FUNCTION "ST10_Flow26_JMagnetLoad&Unload" : Void
VERSION : 1.0
VAR_INPUT
  Enable : BOOL;
END_VAR
VAR_TEMP
  idx : INT;
  tr_cond : ARRAY[1..607] OF BOOL;
  next_active : ARRAY[1..247] OF BOOL;
END_VAR
BEGIN
  IF NOT Enable THEN
    "DB_ST10_Flow26_JMagnetLoad_Unload_State".Flow.Initialized := FALSE;
    FOR idx := 1 TO 247 DO
      "DB_ST10_Flow26_JMagnetLoad_Unload_State".Flow.StepActive[idx] := FALSE;
      "DB_ST10_Flow26_JMagnetLoad_Unload_State".Flow.StepPrev[idx] := FALSE;
    END_FOR;
    "DB_ST10_Flow26_JMagnetLoad_Unload_State".Flow.PalltReleaseRuning := FALSE;
    RETURN;
  END_IF;

  IF NOT "DB_ST10_Flow26_JMagnetLoad_Unload_State".Flow.Initialized THEN
    FOR idx := 1 TO 247 DO
      "DB_ST10_Flow26_JMagnetLoad_Unload_State".Flow.StepActive[idx] := FALSE;
      "DB_ST10_Flow26_JMagnetLoad_Unload_State".Flow.StepPrev[idx] := FALSE;
    END_FOR;
    "DB_ST10_Flow26_JMagnetLoad_Unload_State".Flow.StepActive[1] := TRUE;
    "DB_ST10_Flow26_JMagnetLoad_Unload_State".Flow.StepActive[200] := TRUE;
    "DB_ST10_Flow26_JMagnetLoad_Unload_State".Flow.Initialized := TRUE;
  END_IF;


  IF "DB_ST10_Flow26_JMagnetLoad_Unload_State".Flow.StepActive[119] THEN
    "DB_ST10_Flow26_JMagnetLoad_Unload_State".Flow.StepTime.AriveTimeDelay_1 := "DB_ST10_Flow26_JMagnetLoad_Unload_State".Flow.StepTime.AriveTimeDelay_1 + OB1_PREV_CYCLE;
  ELSE
    "DB_ST10_Flow26_JMagnetLoad_Unload_State".Flow.StepTime.AriveTimeDelay_1 := T#0S;
  END_IF;
  IF "DB_ST10_Flow26_JMagnetLoad_Unload_State".Flow.StepActive[168] THEN
    "DB_ST10_Flow26_JMagnetLoad_Unload_State".Flow.StepTime.AriveTimeDelay_10 := "DB_ST10_Flow26_JMagnetLoad_Unload_State".Flow.StepTime.AriveTimeDelay_10 + OB1_PREV_CYCLE;
  ELSE
    "DB_ST10_Flow26_JMagnetLoad_Unload_State".Flow.StepTime.AriveTimeDelay_10 := T#0S;
  END_IF;
  IF "DB_ST10_Flow26_JMagnetLoad_Unload_State".Flow.StepActive[173] THEN
    "DB_ST10_Flow26_JMagnetLoad_Unload_State".Flow.StepTime.AriveTimeDelay_11 := "DB_ST10_Flow26_JMagnetLoad_Unload_State".Flow.StepTime.AriveTimeDelay_11 + OB1_PREV_CYCLE;
  ELSE
    "DB_ST10_Flow26_JMagnetLoad_Unload_State".Flow.StepTime.AriveTimeDelay_11 := T#0S;
  END_IF;
  IF "DB_ST10_Flow26_JMagnetLoad_Unload_State".Flow.StepActive[120] THEN
    "DB_ST10_Flow26_JMagnetLoad_Unload_State".Flow.StepTime.AriveTimeDelay_2 := "DB_ST10_Flow26_JMagnetLoad_Unload_State".Flow.StepTime.AriveTimeDelay_2 + OB1_PREV_CYCLE;
  ELSE
    "DB_ST10_Flow26_JMagnetLoad_Unload_State".Flow.StepTime.AriveTimeDelay_2 := T#0S;
  END_IF;
  IF "DB_ST10_Flow26_JMagnetLoad_Unload_State".Flow.StepActive[125] THEN
    "DB_ST10_Flow26_JMagnetLoad_Unload_State".Flow.StepTime.AriveTimeDelay_3 := "DB_ST10_Flow26_JMagnetLoad_Unload_State".Flow.StepTime.AriveTimeDelay_3 + OB1_PREV_CYCLE;
  ELSE
    "DB_ST10_Flow26_JMagnetLoad_Unload_State".Flow.StepTime.AriveTimeDelay_3 := T#0S;
  END_IF;
  IF "DB_ST10_Flow26_JMagnetLoad_Unload_State".Flow.StepActive[130] THEN
    "DB_ST10_Flow26_JMagnetLoad_Unload_State".Flow.StepTime.AriveTimeDelay_4 := "DB_ST10_Flow26_JMagnetLoad_Unload_State".Flow.StepTime.AriveTimeDelay_4 + OB1_PREV_CYCLE;
  ELSE
    "DB_ST10_Flow26_JMagnetLoad_Unload_State".Flow.StepTime.AriveTimeDelay_4 := T#0S;
  END_IF;
  IF "DB_ST10_Flow26_JMagnetLoad_Unload_State".Flow.StepActive[136] THEN
    "DB_ST10_Flow26_JMagnetLoad_Unload_State".Flow.StepTime.AriveTimeDelay_5 := "DB_ST10_Flow26_JMagnetLoad_Unload_State".Flow.StepTime.AriveTimeDelay_5 + OB1_PREV_CYCLE;
  ELSE
    "DB_ST10_Flow26_JMagnetLoad_Unload_State".Flow.StepTime.AriveTimeDelay_5 := T#0S;
  END_IF;
  IF "DB_ST10_Flow26_JMagnetLoad_Unload_State".Flow.StepActive[141] THEN
    "DB_ST10_Flow26_JMagnetLoad_Unload_State".Flow.StepTime.AriveTimeDelay_6 := "DB_ST10_Flow26_JMagnetLoad_Unload_State".Flow.StepTime.AriveTimeDelay_6 + OB1_PREV_CYCLE;
  ELSE
    "DB_ST10_Flow26_JMagnetLoad_Unload_State".Flow.StepTime.AriveTimeDelay_6 := T#0S;
  END_IF;
  IF "DB_ST10_Flow26_JMagnetLoad_Unload_State".Flow.StepActive[148] THEN
    "DB_ST10_Flow26_JMagnetLoad_Unload_State".Flow.StepTime.AriveTimeDelay_7 := "DB_ST10_Flow26_JMagnetLoad_Unload_State".Flow.StepTime.AriveTimeDelay_7 + OB1_PREV_CYCLE;
  ELSE
    "DB_ST10_Flow26_JMagnetLoad_Unload_State".Flow.StepTime.AriveTimeDelay_7 := T#0S;
  END_IF;
  IF "DB_ST10_Flow26_JMagnetLoad_Unload_State".Flow.StepActive[159] THEN
    "DB_ST10_Flow26_JMagnetLoad_Unload_State".Flow.StepTime.AriveTimeDelay_8 := "DB_ST10_Flow26_JMagnetLoad_Unload_State".Flow.StepTime.AriveTimeDelay_8 + OB1_PREV_CYCLE;
  ELSE
    "DB_ST10_Flow26_JMagnetLoad_Unload_State".Flow.StepTime.AriveTimeDelay_8 := T#0S;
  END_IF;
  IF "DB_ST10_Flow26_JMagnetLoad_Unload_State".Flow.StepActive[163] THEN
    "DB_ST10_Flow26_JMagnetLoad_Unload_State".Flow.StepTime.AriveTimeDelay_9 := "DB_ST10_Flow26_JMagnetLoad_Unload_State".Flow.StepTime.AriveTimeDelay_9 + OB1_PREV_CYCLE;
  ELSE
    "DB_ST10_Flow26_JMagnetLoad_Unload_State".Flow.StepTime.AriveTimeDelay_9 := T#0S;
  END_IF;
  IF "DB_ST10_Flow26_JMagnetLoad_Unload_State".Flow.StepActive[31] THEN
    "DB_ST10_Flow26_JMagnetLoad_Unload_State".Flow.StepTime.CheckPalletExist := "DB_ST10_Flow26_JMagnetLoad_Unload_State".Flow.StepTime.CheckPalletExist + OB1_PREV_CYCLE;
  ELSE
    "DB_ST10_Flow26_JMagnetLoad_Unload_State".Flow.StepTime.CheckPalletExist := T#0S;
  END_IF;
  IF "DB_ST10_Flow26_JMagnetLoad_Unload_State".Flow.StepActive[32] THEN
    "DB_ST10_Flow26_JMagnetLoad_Unload_State".Flow.StepTime.CheckPalletExist_1 := "DB_ST10_Flow26_JMagnetLoad_Unload_State".Flow.StepTime.CheckPalletExist_1 + OB1_PREV_CYCLE;
  ELSE
    "DB_ST10_Flow26_JMagnetLoad_Unload_State".Flow.StepTime.CheckPalletExist_1 := T#0S;
  END_IF;
  IF "DB_ST10_Flow26_JMagnetLoad_Unload_State".Flow.StepActive[76] THEN
    "DB_ST10_Flow26_JMagnetLoad_Unload_State".Flow.StepTime.CheckPalletExist_10 := "DB_ST10_Flow26_JMagnetLoad_Unload_State".Flow.StepTime.CheckPalletExist_10 + OB1_PREV_CYCLE;
  ELSE
    "DB_ST10_Flow26_JMagnetLoad_Unload_State".Flow.StepTime.CheckPalletExist_10 := T#0S;
  END_IF;
  IF "DB_ST10_Flow26_JMagnetLoad_Unload_State".Flow.StepActive[41] THEN
    "DB_ST10_Flow26_JMagnetLoad_Unload_State".Flow.StepTime.CheckPalletExist_2 := "DB_ST10_Flow26_JMagnetLoad_Unload_State".Flow.StepTime.CheckPalletExist_2 + OB1_PREV_CYCLE;
  ELSE
    "DB_ST10_Flow26_JMagnetLoad_Unload_State".Flow.StepTime.CheckPalletExist_2 := T#0S;
  END_IF;
  IF "DB_ST10_Flow26_JMagnetLoad_Unload_State".Flow.StepActive[45] THEN
    "DB_ST10_Flow26_JMagnetLoad_Unload_State".Flow.StepTime.CheckPalletExist_3 := "DB_ST10_Flow26_JMagnetLoad_Unload_State".Flow.StepTime.CheckPalletExist_3 + OB1_PREV_CYCLE;
  ELSE
    "DB_ST10_Flow26_JMagnetLoad_Unload_State".Flow.StepTime.CheckPalletExist_3 := T#0S;
  END_IF;
  IF "DB_ST10_Flow26_JMagnetLoad_Unload_State".Flow.StepActive[49] THEN
    "DB_ST10_Flow26_JMagnetLoad_Unload_State".Flow.StepTime.CheckPalletExist_4 := "DB_ST10_Flow26_JMagnetLoad_Unload_State".Flow.StepTime.CheckPalletExist_4 + OB1_PREV_CYCLE;
  ELSE
    "DB_ST10_Flow26_JMagnetLoad_Unload_State".Flow.StepTime.CheckPalletExist_4 := T#0S;
  END_IF;
  IF "DB_ST10_Flow26_JMagnetLoad_Unload_State".Flow.StepActive[53] THEN
    "DB_ST10_Flow26_JMagnetLoad_Unload_State".Flow.StepTime.CheckPalletExist_5 := "DB_ST10_Flow26_JMagnetLoad_Unload_State".Flow.StepTime.CheckPalletExist_5 + OB1_PREV_CYCLE;
  ELSE
    "DB_ST10_Flow26_JMagnetLoad_Unload_State".Flow.StepTime.CheckPalletExist_5 := T#0S;
  END_IF;
  IF "DB_ST10_Flow26_JMagnetLoad_Unload_State".Flow.StepActive[57] THEN
    "DB_ST10_Flow26_JMagnetLoad_Unload_State".Flow.StepTime.CheckPalletExist_6 := "DB_ST10_Flow26_JMagnetLoad_Unload_State".Flow.StepTime.CheckPalletExist_6 + OB1_PREV_CYCLE;
  ELSE
    "DB_ST10_Flow26_JMagnetLoad_Unload_State".Flow.StepTime.CheckPalletExist_6 := T#0S;
  END_IF;
  IF "DB_ST10_Flow26_JMagnetLoad_Unload_State".Flow.StepActive[64] THEN
    "DB_ST10_Flow26_JMagnetLoad_Unload_State".Flow.StepTime.CheckPalletExist_7 := "DB_ST10_Flow26_JMagnetLoad_Unload_State".Flow.StepTime.CheckPalletExist_7 + OB1_PREV_CYCLE;
  ELSE
    "DB_ST10_Flow26_JMagnetLoad_Unload_State".Flow.StepTime.CheckPalletExist_7 := T#0S;
  END_IF;
  IF "DB_ST10_Flow26_JMagnetLoad_Unload_State".Flow.StepActive[68] THEN
    "DB_ST10_Flow26_JMagnetLoad_Unload_State".Flow.StepTime.CheckPalletExist_8 := "DB_ST10_Flow26_JMagnetLoad_Unload_State".Flow.StepTime.CheckPalletExist_8 + OB1_PREV_CYCLE;
  ELSE
    "DB_ST10_Flow26_JMagnetLoad_Unload_State".Flow.StepTime.CheckPalletExist_8 := T#0S;
  END_IF;
  IF "DB_ST10_Flow26_JMagnetLoad_Unload_State".Flow.StepActive[72] THEN
    "DB_ST10_Flow26_JMagnetLoad_Unload_State".Flow.StepTime.CheckPalletExist_9 := "DB_ST10_Flow26_JMagnetLoad_Unload_State".Flow.StepTime.CheckPalletExist_9 + OB1_PREV_CYCLE;
  ELSE
    "DB_ST10_Flow26_JMagnetLoad_Unload_State".Flow.StepTime.CheckPalletExist_9 := T#0S;
  END_IF;
  IF "DB_ST10_Flow26_JMagnetLoad_Unload_State".Flow.StepActive[160] THEN
    "DB_ST10_Flow26_JMagnetLoad_Unload_State".Flow.StepTime.LoadStop_11 := "DB_ST10_Flow26_JMagnetLoad_Unload_State".Flow.StepTime.LoadStop_11 + OB1_PREV_CYCLE;
  ELSE
    "DB_ST10_Flow26_JMagnetLoad_Unload_State".Flow.StepTime.LoadStop_11 := T#0S;
  END_IF;
  IF "DB_ST10_Flow26_JMagnetLoad_Unload_State".Flow.StepActive[62] THEN
    "DB_ST10_Flow26_JMagnetLoad_Unload_State".Flow.StepTime.LoadStop_12 := "DB_ST10_Flow26_JMagnetLoad_Unload_State".Flow.StepTime.LoadStop_12 + OB1_PREV_CYCLE;
  ELSE
    "DB_ST10_Flow26_JMagnetLoad_Unload_State".Flow.StepTime.LoadStop_12 := T#0S;
  END_IF;
  IF "DB_ST10_Flow26_JMagnetLoad_Unload_State".Flow.StepActive[63] THEN
    "DB_ST10_Flow26_JMagnetLoad_Unload_State".Flow.StepTime.LoadStop_13 := "DB_ST10_Flow26_JMagnetLoad_Unload_State".Flow.StepTime.LoadStop_13 + OB1_PREV_CYCLE;
  ELSE
    "DB_ST10_Flow26_JMagnetLoad_Unload_State".Flow.StepTime.LoadStop_13 := T#0S;
  END_IF;
  IF "DB_ST10_Flow26_JMagnetLoad_Unload_State".Flow.StepActive[61] THEN
    "DB_ST10_Flow26_JMagnetLoad_Unload_State".Flow.StepTime.LoadStop_14 := "DB_ST10_Flow26_JMagnetLoad_Unload_State".Flow.StepTime.LoadStop_14 + OB1_PREV_CYCLE;
  ELSE
    "DB_ST10_Flow26_JMagnetLoad_Unload_State".Flow.StepTime.LoadStop_14 := T#0S;
  END_IF;
  IF "DB_ST10_Flow26_JMagnetLoad_Unload_State".Flow.StepActive[25] THEN
    "DB_ST10_Flow26_JMagnetLoad_Unload_State".Flow.StepTime.MotorRunDelay := "DB_ST10_Flow26_JMagnetLoad_Unload_State".Flow.StepTime.MotorRunDelay + OB1_PREV_CYCLE;
  ELSE
    "DB_ST10_Flow26_JMagnetLoad_Unload_State".Flow.StepTime.MotorRunDelay := T#0S;
  END_IF;
  IF "DB_ST10_Flow26_JMagnetLoad_Unload_State".Flow.StepActive[26] THEN
    "DB_ST10_Flow26_JMagnetLoad_Unload_State".Flow.StepTime.MotorRunDelay_1 := "DB_ST10_Flow26_JMagnetLoad_Unload_State".Flow.StepTime.MotorRunDelay_1 + OB1_PREV_CYCLE;
  ELSE
    "DB_ST10_Flow26_JMagnetLoad_Unload_State".Flow.StepTime.MotorRunDelay_1 := T#0S;
  END_IF;
  IF "DB_ST10_Flow26_JMagnetLoad_Unload_State".Flow.StepActive[118] THEN
    "DB_ST10_Flow26_JMagnetLoad_Unload_State".Flow.StepTime.StoperRelease_1 := "DB_ST10_Flow26_JMagnetLoad_Unload_State".Flow.StepTime.StoperRelease_1 + OB1_PREV_CYCLE;
  ELSE
    "DB_ST10_Flow26_JMagnetLoad_Unload_State".Flow.StepTime.StoperRelease_1 := T#0S;
  END_IF;
  IF "DB_ST10_Flow26_JMagnetLoad_Unload_State".Flow.StepActive[170] THEN
    "DB_ST10_Flow26_JMagnetLoad_Unload_State".Flow.StepTime.StoperRelease_10 := "DB_ST10_Flow26_JMagnetLoad_Unload_State".Flow.StepTime.StoperRelease_10 + OB1_PREV_CYCLE;
  ELSE
    "DB_ST10_Flow26_JMagnetLoad_Unload_State".Flow.StepTime.StoperRelease_10 := T#0S;
  END_IF;
  IF "DB_ST10_Flow26_JMagnetLoad_Unload_State".Flow.StepActive[175] THEN
    "DB_ST10_Flow26_JMagnetLoad_Unload_State".Flow.StepTime.StoperRelease_11 := "DB_ST10_Flow26_JMagnetLoad_Unload_State".Flow.StepTime.StoperRelease_11 + OB1_PREV_CYCLE;
  ELSE
    "DB_ST10_Flow26_JMagnetLoad_Unload_State".Flow.StepTime.StoperRelease_11 := T#0S;
  END_IF;
  IF "DB_ST10_Flow26_JMagnetLoad_Unload_State".Flow.StepActive[122] THEN
    "DB_ST10_Flow26_JMagnetLoad_Unload_State".Flow.StepTime.StoperRelease_2 := "DB_ST10_Flow26_JMagnetLoad_Unload_State".Flow.StepTime.StoperRelease_2 + OB1_PREV_CYCLE;
  ELSE
    "DB_ST10_Flow26_JMagnetLoad_Unload_State".Flow.StepTime.StoperRelease_2 := T#0S;
  END_IF;
  IF "DB_ST10_Flow26_JMagnetLoad_Unload_State".Flow.StepActive[127] THEN
    "DB_ST10_Flow26_JMagnetLoad_Unload_State".Flow.StepTime.StoperRelease_3 := "DB_ST10_Flow26_JMagnetLoad_Unload_State".Flow.StepTime.StoperRelease_3 + OB1_PREV_CYCLE;
  ELSE
    "DB_ST10_Flow26_JMagnetLoad_Unload_State".Flow.StepTime.StoperRelease_3 := T#0S;
  END_IF;
  IF "DB_ST10_Flow26_JMagnetLoad_Unload_State".Flow.StepActive[133] THEN
    "DB_ST10_Flow26_JMagnetLoad_Unload_State".Flow.StepTime.StoperRelease_4 := "DB_ST10_Flow26_JMagnetLoad_Unload_State".Flow.StepTime.StoperRelease_4 + OB1_PREV_CYCLE;
  ELSE
    "DB_ST10_Flow26_JMagnetLoad_Unload_State".Flow.StepTime.StoperRelease_4 := T#0S;
  END_IF;
  IF "DB_ST10_Flow26_JMagnetLoad_Unload_State".Flow.StepActive[138] THEN
    "DB_ST10_Flow26_JMagnetLoad_Unload_State".Flow.StepTime.StoperRelease_5 := "DB_ST10_Flow26_JMagnetLoad_Unload_State".Flow.StepTime.StoperRelease_5 + OB1_PREV_CYCLE;
  ELSE
    "DB_ST10_Flow26_JMagnetLoad_Unload_State".Flow.StepTime.StoperRelease_5 := T#0S;
  END_IF;
  IF "DB_ST10_Flow26_JMagnetLoad_Unload_State".Flow.StepActive[145] THEN
    "DB_ST10_Flow26_JMagnetLoad_Unload_State".Flow.StepTime.StoperRelease_6 := "DB_ST10_Flow26_JMagnetLoad_Unload_State".Flow.StepTime.StoperRelease_6 + OB1_PREV_CYCLE;
  ELSE
    "DB_ST10_Flow26_JMagnetLoad_Unload_State".Flow.StepTime.StoperRelease_6 := T#0S;
  END_IF;
  IF "DB_ST10_Flow26_JMagnetLoad_Unload_State".Flow.StepActive[150] THEN
    "DB_ST10_Flow26_JMagnetLoad_Unload_State".Flow.StepTime.StoperRelease_7 := "DB_ST10_Flow26_JMagnetLoad_Unload_State".Flow.StepTime.StoperRelease_7 + OB1_PREV_CYCLE;
  ELSE
    "DB_ST10_Flow26_JMagnetLoad_Unload_State".Flow.StepTime.StoperRelease_7 := T#0S;
  END_IF;
  IF "DB_ST10_Flow26_JMagnetLoad_Unload_State".Flow.StepActive[162] THEN
    "DB_ST10_Flow26_JMagnetLoad_Unload_State".Flow.StepTime.StoperRelease_8 := "DB_ST10_Flow26_JMagnetLoad_Unload_State".Flow.StepTime.StoperRelease_8 + OB1_PREV_CYCLE;
  ELSE
    "DB_ST10_Flow26_JMagnetLoad_Unload_State".Flow.StepTime.StoperRelease_8 := T#0S;
  END_IF;
  IF "DB_ST10_Flow26_JMagnetLoad_Unload_State".Flow.StepActive[165] THEN
    "DB_ST10_Flow26_JMagnetLoad_Unload_State".Flow.StepTime.StoperRelease_9 := "DB_ST10_Flow26_JMagnetLoad_Unload_State".Flow.StepTime.StoperRelease_9 + OB1_PREV_CYCLE;
  ELSE
    "DB_ST10_Flow26_JMagnetLoad_Unload_State".Flow.StepTime.StoperRelease_9 := T#0S;
  END_IF;
  IF "DB_ST10_Flow26_JMagnetLoad_Unload_State".Flow.StepActive[116] THEN
    "DB_ST10_Flow26_JMagnetLoad_Unload_State".Flow.StepTime.StoperReset := "DB_ST10_Flow26_JMagnetLoad_Unload_State".Flow.StepTime.StoperReset + OB1_PREV_CYCLE;
  ELSE
    "DB_ST10_Flow26_JMagnetLoad_Unload_State".Flow.StepTime.StoperReset := T#0S;
  END_IF;
  IF "DB_ST10_Flow26_JMagnetLoad_Unload_State".Flow.StepActive[124] THEN
    "DB_ST10_Flow26_JMagnetLoad_Unload_State".Flow.StepTime.TimeDelay := "DB_ST10_Flow26_JMagnetLoad_Unload_State".Flow.StepTime.TimeDelay + OB1_PREV_CYCLE;
  ELSE
    "DB_ST10_Flow26_JMagnetLoad_Unload_State".Flow.StepTime.TimeDelay := T#0S;
  END_IF;
  IF "DB_ST10_Flow26_JMagnetLoad_Unload_State".Flow.StepActive[129] THEN
    "DB_ST10_Flow26_JMagnetLoad_Unload_State".Flow.StepTime.TimeDelay_1 := "DB_ST10_Flow26_JMagnetLoad_Unload_State".Flow.StepTime.TimeDelay_1 + OB1_PREV_CYCLE;
  ELSE
    "DB_ST10_Flow26_JMagnetLoad_Unload_State".Flow.StepTime.TimeDelay_1 := T#0S;
  END_IF;
  IF "DB_ST10_Flow26_JMagnetLoad_Unload_State".Flow.StepActive[135] THEN
    "DB_ST10_Flow26_JMagnetLoad_Unload_State".Flow.StepTime.TimeDelay_2 := "DB_ST10_Flow26_JMagnetLoad_Unload_State".Flow.StepTime.TimeDelay_2 + OB1_PREV_CYCLE;
  ELSE
    "DB_ST10_Flow26_JMagnetLoad_Unload_State".Flow.StepTime.TimeDelay_2 := T#0S;
  END_IF;
  IF "DB_ST10_Flow26_JMagnetLoad_Unload_State".Flow.StepActive[140] THEN
    "DB_ST10_Flow26_JMagnetLoad_Unload_State".Flow.StepTime.TimeDelay_3 := "DB_ST10_Flow26_JMagnetLoad_Unload_State".Flow.StepTime.TimeDelay_3 + OB1_PREV_CYCLE;
  ELSE
    "DB_ST10_Flow26_JMagnetLoad_Unload_State".Flow.StepTime.TimeDelay_3 := T#0S;
  END_IF;
  IF "DB_ST10_Flow26_JMagnetLoad_Unload_State".Flow.StepActive[147] THEN
    "DB_ST10_Flow26_JMagnetLoad_Unload_State".Flow.StepTime.TimeDelay_4 := "DB_ST10_Flow26_JMagnetLoad_Unload_State".Flow.StepTime.TimeDelay_4 + OB1_PREV_CYCLE;
  ELSE
    "DB_ST10_Flow26_JMagnetLoad_Unload_State".Flow.StepTime.TimeDelay_4 := T#0S;
  END_IF;
  IF "DB_ST10_Flow26_JMagnetLoad_Unload_State".Flow.StepActive[152] THEN
    "DB_ST10_Flow26_JMagnetLoad_Unload_State".Flow.StepTime.TimeDelay_5 := "DB_ST10_Flow26_JMagnetLoad_Unload_State".Flow.StepTime.TimeDelay_5 + OB1_PREV_CYCLE;
  ELSE
    "DB_ST10_Flow26_JMagnetLoad_Unload_State".Flow.StepTime.TimeDelay_5 := T#0S;
  END_IF;
  IF "DB_ST10_Flow26_JMagnetLoad_Unload_State".Flow.StepActive[167] THEN
    "DB_ST10_Flow26_JMagnetLoad_Unload_State".Flow.StepTime.TimeDelay_6 := "DB_ST10_Flow26_JMagnetLoad_Unload_State".Flow.StepTime.TimeDelay_6 + OB1_PREV_CYCLE;
  ELSE
    "DB_ST10_Flow26_JMagnetLoad_Unload_State".Flow.StepTime.TimeDelay_6 := T#0S;
  END_IF;
  IF "DB_ST10_Flow26_JMagnetLoad_Unload_State".Flow.StepActive[172] THEN
    "DB_ST10_Flow26_JMagnetLoad_Unload_State".Flow.StepTime.TimeDelay_7 := "DB_ST10_Flow26_JMagnetLoad_Unload_State".Flow.StepTime.TimeDelay_7 + OB1_PREV_CYCLE;
  ELSE
    "DB_ST10_Flow26_JMagnetLoad_Unload_State".Flow.StepTime.TimeDelay_7 := T#0S;
  END_IF;
  IF "DB_ST10_Flow26_JMagnetLoad_Unload_State".Flow.StepActive[177] THEN
    "DB_ST10_Flow26_JMagnetLoad_Unload_State".Flow.StepTime.TimeDelay_8 := "DB_ST10_Flow26_JMagnetLoad_Unload_State".Flow.StepTime.TimeDelay_8 + OB1_PREV_CYCLE;
  ELSE
    "DB_ST10_Flow26_JMagnetLoad_Unload_State".Flow.StepTime.TimeDelay_8 := T#0S;
  END_IF;
  IF "DB_ST10_Flow26_JMagnetLoad_Unload_State".Flow.StepActive[184] THEN
    "DB_ST10_Flow26_JMagnetLoad_Unload_State".Flow.StepTime.TimeDelay_9 := "DB_ST10_Flow26_JMagnetLoad_Unload_State".Flow.StepTime.TimeDelay_9 + OB1_PREV_CYCLE;
  ELSE
    "DB_ST10_Flow26_JMagnetLoad_Unload_State".Flow.StepTime.TimeDelay_9 := T#0S;
  END_IF;

  tr_cond[1] := (TRUE) AND ("DB_ST10_Flow26_JMagnetLoad_Unload_State".Flow.iSysInface.Ready);
  tr_cond[2] := TRUE;
  tr_cond[3] := TRUE;
  tr_cond[10] := TRUE;
  tr_cond[27] := TRUE;
  tr_cond[28] := TRUE;
  tr_cond[29] := ("DB_ST10_Flow26_JMagnetLoad_Unload_State".Flow.StepTime.MotorRunDelay) > (t#5000MS);
  tr_cond[30] := TRUE;
  tr_cond[31] := ("DB_ST10_Flow26_JMagnetLoad_Unload_State".Flow.StepTime.MotorRunDelay_1) > (t#5000MS);
  tr_cond[32] := ("DB_ST10_Flow26_JMagnetLoad_Unload_State".Flow.StepTime.CheckPalletExist_7) > (t#1000MS);
  tr_cond[33] := TRUE;
  tr_cond[34] := (("DB_ST10_Flow26_JMagnetLoad_Unload_State".Flow.StepTime.CheckPalletExist) > (t#1000MS)) AND (NOT ("DB_ST10_Flow26_JMagnetLoad_Unload_State".AutoProcessControl.Robot_1.ClearPart));
  tr_cond[35] := ("DB_ST10_Flow26_JMagnetLoad_Unload_State".Flow.StepTime.CheckPalletExist_1) > (t#1000MS);
  tr_cond[36] := ("DB_ST10_Flow26_JMagnetLoad_Unload_State".Flow.StepTime.CheckPalletExist_2) > (t#1000MS);
  tr_cond[37] := ((TRUE) AND (MotorControl.Dev[13].OutControl.o_Ready)) AND (MotorControl.Dev[14].OutControl.o_Ready);
  tr_cond[38] := TRUE;
  tr_cond[39] := (TRUE) AND (MotorControl.Dev[13].OutControl.o_Ready);
  tr_cond[40] := (TRUE) AND ("DB_ST10_Flow26_JMagnetLoad_Unload_State".AutoProcessControl.Global.J.LoadStopRequestPallet_1);
  tr_cond[41] := ((TRUE) AND (iJ-magnetLoadingDetection2)) OR ((TRUE) AND ("DB_ST10_Flow26_JMagnetLoad_Unload_State".AutoProcessControl.Global.J.EmptyPallet));
  tr_cond[42] := ((TRUE) AND (iJ-magnetLoadingDetection3)) OR ((TRUE) AND ("DB_ST10_Flow26_JMagnetLoad_Unload_State".AutoProcessControl.Global.J.EmptyPallet));
  tr_cond[43] := (TRUE) AND (MotorControl.Dev[13].OutControl.o_Ready);
  tr_cond[44] := (TRUE) AND ("DB_ST10_Flow26_JMagnetLoad_Unload_State".AutoProcessControl.Global.J.LoadStopRequestPallet_2);
  tr_cond[45] := ((TRUE) AND (iJ-magnetLoadingDetection4)) OR ((TRUE) AND ("DB_ST10_Flow26_JMagnetLoad_Unload_State".AutoProcessControl.Global.J.EmptyPallet));
  tr_cond[46] := (TRUE) AND (MotorControl.Dev[13].OutControl.o_Ready);
  tr_cond[47] := (TRUE) AND ("DB_ST10_Flow26_JMagnetLoad_Unload_State".AutoProcessControl.Global.J.LoadStopRequestPallet_3);
  tr_cond[48] := (((TRUE) AND (iJ-magnetLiftingPalletDischargeDetection)) AND (NOT (iJ-MagnetMiddleDetection))) OR ((TRUE) AND ("DB_ST10_Flow26_JMagnetLoad_Unload_State".AutoProcessControl.Global.J.EmptyPallet));
  tr_cond[49] := ("DB_ST10_Flow26_JMagnetLoad_Unload_State".Flow.StepTime.CheckPalletExist_3) > (t#1000MS);
  tr_cond[50] := (TRUE) AND (MotorControl.Dev[13].OutControl.o_Ready);
  tr_cond[51] := (TRUE) AND ("DB_ST10_Flow26_JMagnetLoad_Unload_State".AutoProcessControl.Global.J.LoadStopRequestPallet_4);
  tr_cond[52] := (TRUE) AND (iJ-magnetTakeDetection2);
  tr_cond[53] := ("DB_ST10_Flow26_JMagnetLoad_Unload_State".Flow.StepTime.CheckPalletExist_4) > (t#1000MS);
  tr_cond[54] := (TRUE) AND (MotorControl.Dev[14].OutControl.o_Ready);
  tr_cond[55] := (TRUE) AND ("DB_ST10_Flow26_JMagnetLoad_Unload_State".AutoProcessControl.Global.J.EmptyStopRequestPallet_2);
  tr_cond[56] := (TRUE) AND (iJ-magnetTakeDetection3);
  tr_cond[57] := ("DB_ST10_Flow26_JMagnetLoad_Unload_State".Flow.StepTime.CheckPalletExist_5) > (t#1000MS);
  tr_cond[58] := (TRUE) AND (MotorControl.Dev[14].OutControl.o_Ready);
  tr_cond[59] := (TRUE) AND ("DB_ST10_Flow26_JMagnetLoad_Unload_State".AutoProcessControl.Global.J.EmptyStopRequestPallet_3);
  tr_cond[60] := (TRUE) AND (iJ-magnetTakeShaftDetection);
  tr_cond[61] := ("DB_ST10_Flow26_JMagnetLoad_Unload_State".Flow.StepTime.CheckPalletExist_6) > (t#1000MS);
  tr_cond[62] := (TRUE) AND (MotorControl.Dev[14].OutControl.o_Ready);
  tr_cond[63] := (TRUE) AND (NOT (iJ-magnetTakeShaftDetection));
  tr_cond[64] := ((TRUE) AND (iJ-magnetTakeGateDetection)) OR ((TRUE) AND (NOT ("DB_ST10_Flow26_JMagnetLoad_Unload_State".AutoProcessControl.Global.J.EmptyPallet)));
  tr_cond[65] := ("DB_ST10_Flow26_JMagnetLoad_Unload_State".Flow.StepTime.CheckPalletExist_7) > (t#1000MS);
  tr_cond[66] := (TRUE) AND (MotorControl.Dev[13].OutControl.o_Ready);
  tr_cond[67] := (TRUE) AND (NOT (iJ-magnetTakeGateDetection));
  tr_cond[68] := (TRUE) AND (J-mganePalletEmptyCheck1);
  tr_cond[69] := ("DB_ST10_Flow26_JMagnetLoad_Unload_State".Flow.StepTime.CheckPalletExist_8) > (t#1000MS);
  tr_cond[70] := (TRUE) AND (MotorControl.Dev[13].OutControl.o_Ready);
  tr_cond[71] := (TRUE) AND ("DB_ST10_Flow26_JMagnetLoad_Unload_State".AutoProcessControl.Global.J.LoadStopRequestPallet_2);
  tr_cond[72] := (TRUE) AND (J-mganePalletEmptyCheck2);
  tr_cond[73] := ("DB_ST10_Flow26_JMagnetLoad_Unload_State".Flow.StepTime.CheckPalletExist_9) > (t#1000MS);
  tr_cond[74] := (TRUE) AND (MotorControl.Dev[13].OutControl.o_Ready);
  tr_cond[75] := (TRUE) AND ("DB_ST10_Flow26_JMagnetLoad_Unload_State".AutoProcessControl.Global.J.LoadStopRequestPallet_3);
  tr_cond[76] := (TRUE) AND (J-mganePalletEmptyCheck3);
  tr_cond[77] := ("DB_ST10_Flow26_JMagnetLoad_Unload_State".Flow.StepTime.CheckPalletExist_10) > (t#1000MS);
  tr_cond[78] := (TRUE) AND (MotorControl.Dev[13].OutControl.o_Ready);
  tr_cond[79] := (TRUE) AND ("DB_ST10_Flow26_JMagnetLoad_Unload_State".AutoProcessControl.Global.J.LoadStopRequestPallet_4);
  tr_cond[80] := TRUE;
  tr_cond[81] := (TRUE) AND (NOT (iJ-MagnetMiddleDetection));
  tr_cond[100] := TRUE;
  tr_cond[116] := ("DB_ST10_Flow26_JMagnetLoad_Unload_State".Flow.StepTime.StoperReset) > (t#1000MS);
  tr_cond[117] := TRUE;
  tr_cond[118] := ("DB_ST10_Flow26_JMagnetLoad_Unload_State".Flow.StepTime.StoperRelease_1) > (t#1000MS);
  tr_cond[119] := ("DB_ST10_Flow26_JMagnetLoad_Unload_State".Flow.StepTime.AriveTimeDelay_1) > (t#500MS);
  tr_cond[120] := TRUE;
  tr_cond[121] := TRUE;
  tr_cond[122] := TRUE;
  tr_cond[123] := ("DB_ST10_Flow26_JMagnetLoad_Unload_State".Flow.StepTime.AriveTimeDelay_2) > (t#500MS);
  tr_cond[124] := TRUE;
  tr_cond[125] := ("DB_ST10_Flow26_JMagnetLoad_Unload_State".Flow.StepTime.StoperRelease_2) > (t#1000MS);
  tr_cond[126] := ("DB_ST10_Flow26_JMagnetLoad_Unload_State".Flow.StepTime.CheckPalletExist_1) > (t#1000MS);
  tr_cond[127] := ((TRUE) AND (iJ-magnetLoadingDetection2)) OR ((TRUE) AND ("DB_ST10_Flow26_JMagnetLoad_Unload_State".AutoProcessControl.Global.J.EmptyPallet));
  tr_cond[128] := ("DB_ST10_Flow26_JMagnetLoad_Unload_State".Flow.StepTime.TimeDelay) > (t#500MS);
  tr_cond[129] := ("DB_ST10_Flow26_JMagnetLoad_Unload_State".Flow.StepTime.AriveTimeDelay_3) > (t#500MS);
  tr_cond[130] := TRUE;
  tr_cond[131] := ("DB_ST10_Flow26_JMagnetLoad_Unload_State".Flow.StepTime.StoperRelease_3) > (t#1000MS);
  tr_cond[132] := ("DB_ST10_Flow26_JMagnetLoad_Unload_State".Flow.StepTime.CheckPalletExist_2) > (t#1000MS);
  tr_cond[133] := ((TRUE) AND (iJ-magnetLoadingDetection3)) OR ((TRUE) AND ("DB_ST10_Flow26_JMagnetLoad_Unload_State".AutoProcessControl.Global.J.EmptyPallet));
  tr_cond[134] := ("DB_ST10_Flow26_JMagnetLoad_Unload_State".Flow.StepTime.TimeDelay_1) > (t#500MS);
  tr_cond[135] := TRUE;
  tr_cond[136] := ("DB_ST10_Flow26_JMagnetLoad_Unload_State".Flow.StepTime.AriveTimeDelay_4) > (t#500MS);
  tr_cond[137] := TRUE;
  tr_cond[138] := ("DB_ST10_Flow26_JMagnetLoad_Unload_State".Flow.StepTime.StoperRelease_4) > (t#1000MS);
  tr_cond[139] := ("DB_ST10_Flow26_JMagnetLoad_Unload_State".Flow.StepTime.CheckPalletExist_3) > (t#1000MS);
  tr_cond[140] := ((TRUE) AND (iJ-magnetLoadingDetection4)) OR ((TRUE) AND ("DB_ST10_Flow26_JMagnetLoad_Unload_State".AutoProcessControl.Global.J.EmptyPallet));
  tr_cond[141] := TRUE;
  tr_cond[142] := (TRUE) AND (NOT ("DB_ST10_Flow26_JMagnetLoad_Unload_State".AutoProcessControl.Global.J_EmptyPallet));
  tr_cond[143] := (TRUE) AND ("DB_ST10_Flow26_JMagnetLoad_Unload_State".AutoProcessControl.Global.J_EmptyPallet);
  tr_cond[144] := ("DB_ST10_Flow26_JMagnetLoad_Unload_State".Flow.StepTime.TimeDelay_2) > (t#500MS);
  tr_cond[145] := ("DB_ST10_Flow26_JMagnetLoad_Unload_State".Flow.StepTime.AriveTimeDelay_5) > (t#500MS);
  tr_cond[146] := TRUE;
  tr_cond[147] := ("DB_ST10_Flow26_JMagnetLoad_Unload_State".Flow.StepTime.StoperRelease_5) > (t#1000MS);
  tr_cond[148] := ("DB_ST10_Flow26_JMagnetLoad_Unload_State".Flow.StepTime.CheckPalletExist_4) > (t#1000MS);
  tr_cond[149] := (TRUE) AND (iJ-magnetTakeDetection1);
  tr_cond[150] := ("DB_ST10_Flow26_JMagnetLoad_Unload_State".Flow.StepTime.TimeDelay_3) > (t#500MS);
  tr_cond[151] := ("DB_ST10_Flow26_JMagnetLoad_Unload_State".Flow.StepTime.AriveTimeDelay_6) > (t#500MS);
  tr_cond[152] := TRUE;
  tr_cond[153] := ("DB_ST10_Flow26_JMagnetLoad_Unload_State".Flow.StepTime.StoperRelease_6) > (t#1000MS);
  tr_cond[154] := ("DB_ST10_Flow26_JMagnetLoad_Unload_State".Flow.StepTime.CheckPalletExist_5) > (t#1000MS);
  tr_cond[155] := (TRUE) AND (iJ-magnetTakeDetection2);
  tr_cond[156] := ("DB_ST10_Flow26_JMagnetLoad_Unload_State".Flow.StepTime.TimeDelay_4) > (t#500MS);
  tr_cond[157] := ("DB_ST10_Flow26_JMagnetLoad_Unload_State".Flow.StepTime.AriveTimeDelay_7) > (t#500MS);
  tr_cond[158] := TRUE;
  tr_cond[159] := ("DB_ST10_Flow26_JMagnetLoad_Unload_State".Flow.StepTime.StoperRelease_7) > (t#1000MS);
  tr_cond[160] := ("DB_ST10_Flow26_JMagnetLoad_Unload_State".Flow.StepTime.CheckPalletExist_6) > (t#1000MS);
  tr_cond[161] := (TRUE) AND (iJ-magnetTakeDetection3);
  tr_cond[162] := ("DB_ST10_Flow26_JMagnetLoad_Unload_State".Flow.StepTime.TimeDelay_5) > (t#500MS);
  tr_cond[163] := TRUE;
  tr_cond[164] := (TRUE) AND (NOT ("DB_ST10_Flow26_JMagnetLoad_Unload_State".AutoProcessControl.Global.J.EmptyPallet));
  tr_cond[165] := (TRUE) AND (NOT ("DB_ST10_Flow26_JMagnetLoad_Unload_State".AutoProcessControl.Global.J.EmptyPallet));
  tr_cond[166] := (TRUE) AND (NOT ("DB_ST10_Flow26_JMagnetLoad_Unload_State".AutoProcessControl.Global.J.EmptyPallet));
  tr_cond[167] := (TRUE) AND (NOT ("DB_ST10_Flow26_JMagnetLoad_Unload_State".AutoProcessControl.Global.J.EmptyPallet));
  tr_cond[168] := ("DB_ST10_Flow26_JMagnetLoad_Unload_State".Flow.StepTime.AriveTimeDelay_8) > (t#500MS);
  tr_cond[169] := ("DB_ST10_Flow26_JMagnetLoad_Unload_State".Flow.StepTime.LoadStop_12) > (t#2S);
  tr_cond[170] := ("DB_ST10_Flow26_JMagnetLoad_Unload_State".Flow.StepTime.LoadStop_13) > (t#2S);
  tr_cond[171] := (TRUE) AND ("DB_ST10_Flow26_JMagnetLoad_Unload_State".AutoProcessControl.Global.J.EmptyPallet);
  tr_cond[172] := ("DB_ST10_Flow26_JMagnetLoad_Unload_State".Flow.StepTime.LoadStop_11) > (t#2S);
  tr_cond[173] := TRUE;
  tr_cond[174] := ("DB_ST10_Flow26_JMagnetLoad_Unload_State".Flow.StepTime.StoperRelease_8) > (t#1000MS);
  tr_cond[175] := ("DB_ST10_Flow26_JMagnetLoad_Unload_State".Flow.StepTime.LoadStop_14) > (t#2S);
  tr_cond[176] := ("DB_ST10_Flow26_JMagnetLoad_Unload_State".Flow.StepTime.AriveTimeDelay_9) > (t#500MS);
  tr_cond[177] := TRUE;
  tr_cond[178] := ("DB_ST10_Flow26_JMagnetLoad_Unload_State".Flow.StepTime.StoperRelease_9) > (t#1000MS);
  tr_cond[179] := ("DB_ST10_Flow26_JMagnetLoad_Unload_State".Flow.StepTime.CheckPalletExist_8) > (t#1000MS);
  tr_cond[180] := ((TRUE) AND (J-mganePalletEmptyCheck2)) OR ((TRUE) AND (NOT ("DB_ST10_Flow26_JMagnetLoad_Unload_State".AutoProcessControl.Global.J.EmptyPallet)));
  tr_cond[181] := ("DB_ST10_Flow26_JMagnetLoad_Unload_State".Flow.StepTime.TimeDelay_6) > (t#500MS);
  tr_cond[182] := ("DB_ST10_Flow26_JMagnetLoad_Unload_State".Flow.StepTime.AriveTimeDelay_10) > (t#500MS);
  tr_cond[183] := TRUE;
  tr_cond[184] := ("DB_ST10_Flow26_JMagnetLoad_Unload_State".Flow.StepTime.StoperRelease_10) > (t#1000MS);
  tr_cond[185] := ("DB_ST10_Flow26_JMagnetLoad_Unload_State".Flow.StepTime.CheckPalletExist_9) > (t#1000MS);
  tr_cond[186] := ((TRUE) AND (J-mganePalletEmptyCheck3)) OR ((TRUE) AND (NOT ("DB_ST10_Flow26_JMagnetLoad_Unload_State".AutoProcessControl.Global.J.EmptyPallet)));
  tr_cond[187] := ("DB_ST10_Flow26_JMagnetLoad_Unload_State".Flow.StepTime.TimeDelay_7) > (t#500MS);
  tr_cond[188] := ("DB_ST10_Flow26_JMagnetLoad_Unload_State".Flow.StepTime.AriveTimeDelay_11) > (t#500MS);
  tr_cond[189] := TRUE;
  tr_cond[190] := ("DB_ST10_Flow26_JMagnetLoad_Unload_State".Flow.StepTime.StoperRelease_11) > (t#1000MS);
  tr_cond[191] := ("DB_ST10_Flow26_JMagnetLoad_Unload_State".Flow.StepTime.CheckPalletExist_10) > (t#1000MS);
  tr_cond[192] := (((TRUE) AND (J-mganePalletEmptyCheck4)) AND (iJ-MagnetMiddleDetection)) OR ((TRUE) AND (NOT ("DB_ST10_Flow26_JMagnetLoad_Unload_State".AutoProcessControl.Global.J.EmptyPallet)));
  tr_cond[193] := ("DB_ST10_Flow26_JMagnetLoad_Unload_State".Flow.StepTime.TimeDelay_8) > (t#500MS);
  tr_cond[194] := (TRUE) AND ("DB_ST10_Flow26_JMagnetLoad_Unload_State".AutoProcessControl.Global.J.EmptyPallet);
  tr_cond[195] := (TRUE) AND ("DB_ST10_Flow26_JMagnetLoad_Unload_State".AutoProcessControl.Global.J.EmptyPallet);
  tr_cond[196] := (TRUE) AND ("DB_ST10_Flow26_JMagnetLoad_Unload_State".AutoProcessControl.Global.J.EmptyPallet);
  tr_cond[197] := ((((((((TRUE) AND (ST10Cylinder.Cy[33].Inout.AutoGoHome)) AND (NOT (ST10Cylinder.Cy[33].Inout.AutoGoWork))) AND (ST10Cylinder.Cy[34].Inout.AutoGoHome)) AND (NOT (ST10Cylinder.Cy[34].Inout.AutoGoWork))) AND (ST10Cylinder.Cy[35].Inout.AutoGoHome)) AND (NOT (ST10Cylinder.Cy[35].Inout.AutoGoWork))) AND (ST10Cylinder.Cy[36].Inout.AutoGoHome)) AND (NOT (ST10Cylinder.Cy[36].Inout.AutoGoWork));
  tr_cond[198] := TRUE;
  tr_cond[199] := ((TRUE) AND (J-mganePalletEmptyCheck1)) OR ((TRUE) AND (NOT ("DB_ST10_Flow26_JMagnetLoad_Unload_State".AutoProcessControl.Global.J.EmptyPallet)));
  tr_cond[200] := (TRUE) AND ("DB_ST10_Flow26_JMagnetLoad_Unload_State".AutoProcessControl.Global.J.EmptyPallet);
  tr_cond[201] := ("DB_ST10_Flow26_JMagnetLoad_Unload_State".Flow.StepTime.TimeDelay_9) > (t#500MS);
  tr_cond[202] := TRUE;
  tr_cond[203] := TRUE;
  tr_cond[204] := (TRUE) AND ("DB_ST10_Flow26_JMagnetLoad_Unload_State".AutoProcessControl.Global.J.EmptyPallet);
  tr_cond[205] := (TRUE) AND ("DB_ST10_Flow26_JMagnetLoad_Unload_State".AutoProcessControl.Global.J.EmptyPallet);
  tr_cond[206] := (TRUE) AND ("DB_ST10_Flow26_JMagnetLoad_Unload_State".AutoProcessControl.Global.J.EmptyPallet);
  tr_cond[207] := (TRUE) AND ("DB_ST10_Flow26_JMagnetLoad_Unload_State".AutoProcessControl.Global.J.EmptyPallet);
  tr_cond[249] := TRUE;
  tr_cond[250] := TRUE;
  tr_cond[251] := TRUE;
  tr_cond[252] := TRUE;
  tr_cond[253] := TRUE;
  tr_cond[254] := TRUE;
  tr_cond[255] := TRUE;
  tr_cond[256] := TRUE;
  tr_cond[257] := TRUE;
  tr_cond[258] := TRUE;
  tr_cond[259] := TRUE;
  tr_cond[607] := TRUE;

  FOR idx := 1 TO 247 DO
    next_active[idx] := "DB_ST10_Flow26_JMagnetLoad_Unload_State".Flow.StepActive[idx];
  END_FOR;

  IF "DB_ST10_Flow26_JMagnetLoad_Unload_State".Flow.StepActive[1] THEN
    // Step 1: F26_Initial
    IF NOT "DB_ST10_Flow26_JMagnetLoad_Unload_State".Flow.StepPrev[1] THEN
      #ioPM_Inface.InitialRun := TRUE;
      #ioPM_Inface.InitialOK := FALSE;
      #ioPM_Inface.WaitRunning := FALSE;
      #ioPM_Inface.Running := FALSE;
      #ioPM_Inface.ProcessComplete := FALSE;
      #ioPM_Inface.UnPause := FALSE;
      "Station_Sys".Cmd.Calibration := FALSE;
      "Station_Sys".Cmd.ChangeOver := FALSE;
      "Station_Sys".Cmd.Reserve := FALSE;
      "Station_Sys".Cmd.OneCycle := FALSE;
    END_IF;
    IF tr_cond[1] THEN
      next_active[1] := FALSE;
      next_active[2] := TRUE;
    END_IF;
  END_IF;

  IF "DB_ST10_Flow26_JMagnetLoad_Unload_State".Flow.StepActive[2] THEN
    // Step 2: S2
    IF tr_cond[2] THEN
      next_active[2] := FALSE;
      next_active[3] := TRUE;
    END_IF;
  END_IF;

  IF "DB_ST10_Flow26_JMagnetLoad_Unload_State".Flow.StepActive[3] THEN
    // Step 3: S3
    IF tr_cond[607] THEN
      next_active[3] := FALSE;
      next_active[4] := TRUE;
    END_IF;
  END_IF;

  IF "DB_ST10_Flow26_JMagnetLoad_Unload_State".Flow.StepActive[4] THEN
    // Step 4: S4
    IF tr_cond[3] THEN
      next_active[4] := FALSE;
      next_active[33] := TRUE;
    END_IF;
  END_IF;

  IF "DB_ST10_Flow26_JMagnetLoad_Unload_State".Flow.StepActive[10] THEN
    // Step 10: S10_InitialFinish
    IF NOT "DB_ST10_Flow26_JMagnetLoad_Unload_State".Flow.StepPrev[10] THEN
      #ioPM_Inface.InitialOK := TRUE;
    END_IF;
    IF tr_cond[10] THEN
      next_active[10] := FALSE;
      next_active[100] := TRUE;
    END_IF;
  END_IF;

  IF "DB_ST10_Flow26_JMagnetLoad_Unload_State".Flow.StepActive[23] THEN
    // Step 23: MotorCWStart
    IF NOT "DB_ST10_Flow26_JMagnetLoad_Unload_State".Flow.StepPrev[23] THEN
      "MotorControl".Dev[13].Auto.CCWStart := FALSE;
      "MotorControl".Dev[13].Auto.Start := TRUE;
      "MotorControl".Dev[14].Auto.CCWStart := FALSE;
      "MotorControl".Dev[14].Auto.Start := TRUE;
    END_IF;
    IF tr_cond[27] THEN
      next_active[23] := FALSE;
      next_active[26] := TRUE;
    END_IF;
  END_IF;

  IF "DB_ST10_Flow26_JMagnetLoad_Unload_State".Flow.StepActive[24] THEN
    // Step 24: MotorCWStart_1
    IF NOT "DB_ST10_Flow26_JMagnetLoad_Unload_State".Flow.StepPrev[24] THEN
      "MotorControl".Dev[13].Auto.CCWStart := TRUE;
      "MotorControl".Dev[13].Auto.Start := FALSE;
      "MotorControl".Dev[14].Auto.CCWStart := FALSE;
      "MotorControl".Dev[14].Auto.Start := TRUE;
    END_IF;
    IF tr_cond[28] THEN
      next_active[24] := FALSE;
      next_active[25] := TRUE;
    END_IF;
  END_IF;

  IF "DB_ST10_Flow26_JMagnetLoad_Unload_State".Flow.StepActive[25] THEN
    // Step 25: MotorRunDelay
    IF tr_cond[29] THEN
      next_active[25] := FALSE;
    END_IF;
  END_IF;

  IF "DB_ST10_Flow26_JMagnetLoad_Unload_State".Flow.StepActive[26] THEN
    // Step 26: MotorRunDelay_1
    IF tr_cond[31] THEN
      next_active[26] := FALSE;
      next_active[81] := TRUE;
    END_IF;
  END_IF;

  IF "DB_ST10_Flow26_JMagnetLoad_Unload_State".Flow.StepActive[27] THEN
    // Step 27: StopProcess
    IF tr_cond[33] THEN
      next_active[27] := FALSE;
    END_IF;
  END_IF;

  IF "DB_ST10_Flow26_JMagnetLoad_Unload_State".Flow.StepActive[28] THEN
    // Step 28: LoadingStop_2
    IF tr_cond[120] THEN
      next_active[28] := FALSE;
      next_active[32] := TRUE;
    END_IF;
  END_IF;

  IF "DB_ST10_Flow26_JMagnetLoad_Unload_State".Flow.StepActive[29] THEN
    // Step 29: LoadingStop_3
    IF tr_cond[121] THEN
      next_active[29] := FALSE;
      next_active[41] := TRUE;
    END_IF;
  END_IF;

  IF "DB_ST10_Flow26_JMagnetLoad_Unload_State".Flow.StepActive[30] THEN
    // Step 30: LoadingStop_4
    IF tr_cond[122] THEN
      next_active[30] := FALSE;
      next_active[45] := TRUE;
    END_IF;
  END_IF;

  IF "DB_ST10_Flow26_JMagnetLoad_Unload_State".Flow.StepActive[31] THEN
    // Step 31: CheckPalletExist
    IF NOT "DB_ST10_Flow26_JMagnetLoad_Unload_State".Flow.StepPrev[31] THEN
      "MotorControl".Dev[13].Auto.CCWStart := FALSE;
    END_IF;
    IF tr_cond[34] THEN
      next_active[31] := FALSE;
      next_active[35] := TRUE;
    END_IF;
  END_IF;

  IF "DB_ST10_Flow26_JMagnetLoad_Unload_State".Flow.StepActive[32] THEN
    // Step 32: CheckPalletExist_1
  END_IF;

  IF "DB_ST10_Flow26_JMagnetLoad_Unload_State".Flow.StepActive[33] THEN
    // Step 33: CheckMaterialDoorLock
    IF tr_cond[37] THEN
      next_active[33] := FALSE;
      next_active[143] := TRUE;
    END_IF;
  END_IF;

  IF "DB_ST10_Flow26_JMagnetLoad_Unload_State".Flow.StepActive[34] THEN
    // Step 34: MotorRun
    IF NOT "DB_ST10_Flow26_JMagnetLoad_Unload_State".Flow.StepPrev[34] THEN
      "MotorControl".Dev[13].Auto.Start := TRUE;
      "MotorControl".Dev[13].Auto.CCWStart := FALSE;
      "MotorControl".Dev[14].Auto.Start := TRUE;
      "MotorControl".Dev[14].Auto.CCWStart := FALSE;
    END_IF;
    IF tr_cond[38] THEN
      next_active[34] := FALSE;
      next_active[27] := TRUE;
    END_IF;
  END_IF;

  IF "DB_ST10_Flow26_JMagnetLoad_Unload_State".Flow.StepActive[35] THEN
    // Step 35: WaitLineMotorReady
    IF tr_cond[39] THEN
      next_active[35] := FALSE;
      next_active[36] := TRUE;
    END_IF;
  END_IF;

  IF "DB_ST10_Flow26_JMagnetLoad_Unload_State".Flow.StepActive[36] THEN
    // Step 36: WaitPalletRequestRelease
  END_IF;

  IF "DB_ST10_Flow26_JMagnetLoad_Unload_State".Flow.StepActive[37] THEN
    // Step 37: WaitPalletArrveNextPos
    IF NOT "DB_ST10_Flow26_JMagnetLoad_Unload_State".Flow.StepPrev[37] THEN
      "MotorControl".Dev[13].Auto.Start := TRUE;
      "MotorControl".Dev[13].Auto.CCWStart := FALSE;
    END_IF;
    IF tr_cond[41] THEN
      next_active[37] := FALSE;
      next_active[119] := TRUE;
    END_IF;
  END_IF;

  IF "DB_ST10_Flow26_JMagnetLoad_Unload_State".Flow.StepActive[38] THEN
    // Step 38: WaitLineMotorReady_1
    IF tr_cond[43] THEN
      next_active[38] := FALSE;
      next_active[39] := TRUE;
    END_IF;
  END_IF;

  IF "DB_ST10_Flow26_JMagnetLoad_Unload_State".Flow.StepActive[39] THEN
    // Step 39: WaitPalletRequestRelease_1
  END_IF;

  IF "DB_ST10_Flow26_JMagnetLoad_Unload_State".Flow.StepActive[40] THEN
    // Step 40: WaitPalletArrveNextPos_1
    IF NOT "DB_ST10_Flow26_JMagnetLoad_Unload_State".Flow.StepPrev[40] THEN
      "MotorControl".Dev[13].Auto.Start := TRUE;
      "MotorControl".Dev[13].Auto.CCWStart := FALSE;
    END_IF;
    IF tr_cond[42] THEN
      next_active[40] := FALSE;
      next_active[120] := TRUE;
    END_IF;
  END_IF;

  IF "DB_ST10_Flow26_JMagnetLoad_Unload_State".Flow.StepActive[41] THEN
    // Step 41: CheckPalletExist_2
  END_IF;

  IF "DB_ST10_Flow26_JMagnetLoad_Unload_State".Flow.StepActive[42] THEN
    // Step 42: WaitLineMotorReady_2
    IF tr_cond[46] THEN
      next_active[42] := FALSE;
      next_active[43] := TRUE;
    END_IF;
  END_IF;

  IF "DB_ST10_Flow26_JMagnetLoad_Unload_State".Flow.StepActive[43] THEN
    // Step 43: WaitPalletRequestRelease_2
  END_IF;

  IF "DB_ST10_Flow26_JMagnetLoad_Unload_State".Flow.StepActive[44] THEN
    // Step 44: WaitPalletArrveNextPos_2
    IF NOT "DB_ST10_Flow26_JMagnetLoad_Unload_State".Flow.StepPrev[44] THEN
      "MotorControl".Dev[13].Auto.Start := TRUE;
      "MotorControl".Dev[13].Auto.CCWStart := FALSE;
    END_IF;
    IF tr_cond[45] THEN
      next_active[44] := FALSE;
      next_active[125] := TRUE;
    END_IF;
  END_IF;

  IF "DB_ST10_Flow26_JMagnetLoad_Unload_State".Flow.StepActive[45] THEN
    // Step 45: CheckPalletExist_3
  END_IF;

  IF "DB_ST10_Flow26_JMagnetLoad_Unload_State".Flow.StepActive[46] THEN
    // Step 46: WaitLineMotorReady_3
    IF tr_cond[50] THEN
      next_active[46] := FALSE;
      next_active[47] := TRUE;
    END_IF;
  END_IF;

  IF "DB_ST10_Flow26_JMagnetLoad_Unload_State".Flow.StepActive[47] THEN
    // Step 47: WaitPalletRequestRelease_3
  END_IF;

  IF "DB_ST10_Flow26_JMagnetLoad_Unload_State".Flow.StepActive[48] THEN
    // Step 48: WaitPalletArrveNextPos_3
    IF NOT "DB_ST10_Flow26_JMagnetLoad_Unload_State".Flow.StepPrev[48] THEN
      "MotorControl".Dev[13].Auto.Start := TRUE;
      "MotorControl".Dev[13].Auto.CCWStart := FALSE;
      "MotorControl".Dev[2].Auto.CCWStart := FALSE;
      "MotorControl".Dev[2].Auto.Start := TRUE;
    END_IF;
    IF tr_cond[48] THEN
      next_active[48] := FALSE;
      next_active[130] := TRUE;
    END_IF;
  END_IF;

  IF "DB_ST10_Flow26_JMagnetLoad_Unload_State".Flow.StepActive[49] THEN
    // Step 49: CheckPalletExist_4
  END_IF;

  IF "DB_ST10_Flow26_JMagnetLoad_Unload_State".Flow.StepActive[50] THEN
    // Step 50: WaitLineMotorReady_4
    IF tr_cond[54] THEN
      next_active[50] := FALSE;
      next_active[51] := TRUE;
    END_IF;
  END_IF;

  IF "DB_ST10_Flow26_JMagnetLoad_Unload_State".Flow.StepActive[51] THEN
    // Step 51: WaitPalletRequestRelease_4
    IF tr_cond[55] THEN
      next_active[51] := FALSE;
      next_active[138] := TRUE;
    END_IF;
  END_IF;

  IF "DB_ST10_Flow26_JMagnetLoad_Unload_State".Flow.StepActive[52] THEN
    // Step 52: WaitPalletArrveNextPos_4
    IF NOT "DB_ST10_Flow26_JMagnetLoad_Unload_State".Flow.StepPrev[52] THEN
      "MotorControl".Dev[14].Auto.Start := TRUE;
      "MotorControl".Dev[14].Auto.CCWStart := FALSE;
    END_IF;
    IF tr_cond[52] THEN
      next_active[52] := FALSE;
      next_active[136] := TRUE;
    END_IF;
  END_IF;

  IF "DB_ST10_Flow26_JMagnetLoad_Unload_State".Flow.StepActive[53] THEN
    // Step 53: CheckPalletExist_5
  END_IF;

  IF "DB_ST10_Flow26_JMagnetLoad_Unload_State".Flow.StepActive[54] THEN
    // Step 54: WaitLineMotorReady_5
    IF tr_cond[58] THEN
      next_active[54] := FALSE;
      next_active[55] := TRUE;
    END_IF;
  END_IF;

  IF "DB_ST10_Flow26_JMagnetLoad_Unload_State".Flow.StepActive[55] THEN
    // Step 55: WaitPalletRequestRelease_5
    IF tr_cond[59] THEN
      next_active[55] := FALSE;
      next_active[145] := TRUE;
    END_IF;
  END_IF;

  IF "DB_ST10_Flow26_JMagnetLoad_Unload_State".Flow.StepActive[56] THEN
    // Step 56: WaitPalletArrveNextPos_5
    IF NOT "DB_ST10_Flow26_JMagnetLoad_Unload_State".Flow.StepPrev[56] THEN
      "MotorControl".Dev[14].Auto.Start := TRUE;
      "MotorControl".Dev[14].Auto.CCWStart := FALSE;
    END_IF;
    IF tr_cond[56] THEN
      next_active[56] := FALSE;
      next_active[141] := TRUE;
    END_IF;
  END_IF;

  IF "DB_ST10_Flow26_JMagnetLoad_Unload_State".Flow.StepActive[57] THEN
    // Step 57: CheckPalletExist_6
  END_IF;

  IF "DB_ST10_Flow26_JMagnetLoad_Unload_State".Flow.StepActive[58] THEN
    // Step 58: WaitLineMotorReady_6
    IF tr_cond[62] THEN
      next_active[58] := FALSE;
      next_active[59] := TRUE;
    END_IF;
  END_IF;

  IF "DB_ST10_Flow26_JMagnetLoad_Unload_State".Flow.StepActive[59] THEN
    // Step 59: WaitPalletRequestRelease_6
    IF tr_cond[63] THEN
      next_active[59] := FALSE;
      next_active[150] := TRUE;
    END_IF;
  END_IF;

  IF "DB_ST10_Flow26_JMagnetLoad_Unload_State".Flow.StepActive[60] THEN
    // Step 60: WaitPalletArrveNextPos_6
    IF NOT "DB_ST10_Flow26_JMagnetLoad_Unload_State".Flow.StepPrev[60] THEN
      "MotorControl".Dev[14].Auto.Start := TRUE;
      "MotorControl".Dev[14].Auto.CCWStart := FALSE;
    END_IF;
    IF tr_cond[60] THEN
      next_active[60] := FALSE;
      next_active[148] := TRUE;
    END_IF;
  END_IF;

  IF "DB_ST10_Flow26_JMagnetLoad_Unload_State".Flow.StepActive[61] THEN
    // Step 61: LoadStop_14
    IF tr_cond[175] THEN
      next_active[61] := FALSE;
      next_active[76] := TRUE;
    END_IF;
  END_IF;

  IF "DB_ST10_Flow26_JMagnetLoad_Unload_State".Flow.StepActive[62] THEN
    // Step 62: LoadStop_12
    IF tr_cond[169] THEN
      next_active[62] := FALSE;
      next_active[68] := TRUE;
    END_IF;
  END_IF;

  IF "DB_ST10_Flow26_JMagnetLoad_Unload_State".Flow.StepActive[63] THEN
    // Step 63: LoadStop_13
    IF tr_cond[170] THEN
      next_active[63] := FALSE;
      next_active[72] := TRUE;
    END_IF;
  END_IF;

  IF "DB_ST10_Flow26_JMagnetLoad_Unload_State".Flow.StepActive[64] THEN
    // Step 64: CheckPalletExist_7
  END_IF;

  IF "DB_ST10_Flow26_JMagnetLoad_Unload_State".Flow.StepActive[65] THEN
    // Step 65: WaitLineMotorReady_7
    IF tr_cond[66] THEN
      next_active[65] := FALSE;
      next_active[66] := TRUE;
    END_IF;
  END_IF;

  IF "DB_ST10_Flow26_JMagnetLoad_Unload_State".Flow.StepActive[66] THEN
    // Step 66: WaitPalletRequestRelease_7
    IF tr_cond[67] THEN
      next_active[66] := FALSE;
      next_active[162] := TRUE;
    END_IF;
  END_IF;

  IF "DB_ST10_Flow26_JMagnetLoad_Unload_State".Flow.StepActive[67] THEN
    // Step 67: WaitPalletArrveNextPos_7
    IF tr_cond[64] THEN
      next_active[67] := FALSE;
      next_active[159] := TRUE;
    END_IF;
  END_IF;

  IF "DB_ST10_Flow26_JMagnetLoad_Unload_State".Flow.StepActive[68] THEN
    // Step 68: CheckPalletExist_8
  END_IF;

  IF "DB_ST10_Flow26_JMagnetLoad_Unload_State".Flow.StepActive[69] THEN
    // Step 69: WaitLineMotorReady_8
    IF tr_cond[70] THEN
      next_active[69] := FALSE;
      next_active[70] := TRUE;
    END_IF;
  END_IF;

  IF "DB_ST10_Flow26_JMagnetLoad_Unload_State".Flow.StepActive[70] THEN
    // Step 70: WaitPalletRequestRelease_8
    IF tr_cond[71] THEN
      next_active[70] := FALSE;
      next_active[165] := TRUE;
    END_IF;
  END_IF;

  IF "DB_ST10_Flow26_JMagnetLoad_Unload_State".Flow.StepActive[71] THEN
    // Step 71: WaitPalletArrveNextPos_8
    IF tr_cond[68] THEN
      next_active[71] := FALSE;
      next_active[163] := TRUE;
    END_IF;
  END_IF;

  IF "DB_ST10_Flow26_JMagnetLoad_Unload_State".Flow.StepActive[72] THEN
    // Step 72: CheckPalletExist_9
  END_IF;

  IF "DB_ST10_Flow26_JMagnetLoad_Unload_State".Flow.StepActive[73] THEN
    // Step 73: WaitLineMotorReady_9
    IF tr_cond[74] THEN
      next_active[73] := FALSE;
      next_active[74] := TRUE;
    END_IF;
  END_IF;

  IF "DB_ST10_Flow26_JMagnetLoad_Unload_State".Flow.StepActive[74] THEN
    // Step 74: WaitPalletRequestRelease_9
    IF tr_cond[75] THEN
      next_active[74] := FALSE;
      next_active[170] := TRUE;
    END_IF;
  END_IF;

  IF "DB_ST10_Flow26_JMagnetLoad_Unload_State".Flow.StepActive[75] THEN
    // Step 75: WaitPalletArrveNextPos_9
    IF tr_cond[72] THEN
      next_active[75] := FALSE;
      next_active[168] := TRUE;
    END_IF;
  END_IF;

  IF "DB_ST10_Flow26_JMagnetLoad_Unload_State".Flow.StepActive[76] THEN
    // Step 76: CheckPalletExist_10
  END_IF;

  IF "DB_ST10_Flow26_JMagnetLoad_Unload_State".Flow.StepActive[77] THEN
    // Step 77: WaitLineMotorReady_10
    IF tr_cond[78] THEN
      next_active[77] := FALSE;
      next_active[78] := TRUE;
    END_IF;
  END_IF;

  IF "DB_ST10_Flow26_JMagnetLoad_Unload_State".Flow.StepActive[78] THEN
    // Step 78: WaitPalletRequestRelease_10
    IF tr_cond[79] THEN
      next_active[78] := FALSE;
      next_active[175] := TRUE;
    END_IF;
  END_IF;

  IF "DB_ST10_Flow26_JMagnetLoad_Unload_State".Flow.StepActive[79] THEN
    // Step 79: WaitPalletArrveNextPos_10
    IF tr_cond[76] THEN
      next_active[79] := FALSE;
      next_active[173] := TRUE;
    END_IF;
  END_IF;

  IF "DB_ST10_Flow26_JMagnetLoad_Unload_State".Flow.StepActive[80] THEN
    // Step 80: MotorRun_1
    IF NOT "DB_ST10_Flow26_JMagnetLoad_Unload_State".Flow.StepPrev[80] THEN
      "MotorControl".Dev[13].Auto.Start := FALSE;
      "MotorControl".Dev[13].Auto.CCWStart := TRUE;
      "MotorControl".Dev[14].Auto.Start := TRUE;
      "MotorControl".Dev[14].Auto.CCWStart := FALSE;
    END_IF;
    IF tr_cond[80] THEN
      next_active[80] := FALSE;
      next_active[182] := TRUE;
    END_IF;
  END_IF;

  IF "DB_ST10_Flow26_JMagnetLoad_Unload_State".Flow.StepActive[81] THEN
    // Step 81: MiddleNoPallet?
    IF tr_cond[81] THEN
      next_active[81] := FALSE;
    END_IF;
  END_IF;

  IF "DB_ST10_Flow26_JMagnetLoad_Unload_State".Flow.StepActive[100] THEN
    // Step 100: ProcessStart
    IF NOT "DB_ST10_Flow26_JMagnetLoad_Unload_State".Flow.StepPrev[100] THEN
      #ioPM_Inface.InitialRun := FALSE;
      #ioPM_Inface.ProcessComplete := FALSE;
      #ioPM_Inface.ProcessStart := FALSE;
      #ioPM_Inface.InitialOK := TRUE;
      #ioPM_Inface.WaitRunning := TRUE;
      #ioPM_Inface.ProcessResult:=0;
    END_IF;
    IF tr_cond[100] THEN
      next_active[100] := FALSE;
      next_active[34] := TRUE;
    END_IF;
  END_IF;

  IF "DB_ST10_Flow26_JMagnetLoad_Unload_State".Flow.StepActive[116] THEN
    // Step 116: StoperReset
    IF NOT "DB_ST10_Flow26_JMagnetLoad_Unload_State".Flow.StepPrev[116] THEN
      "ST10Cylinder".Cy[33].Inout.AutoGoHome := TRUE;
      "ST10Cylinder".Cy[33].Inout.AutoGoWork := FALSE;
      "ST10Cylinder".Cy[34].Inout.AutoGoHome := TRUE;
      "ST10Cylinder".Cy[34].Inout.AutoGoWork := FALSE;
      "ST10Cylinder".Cy[35].Inout.AutoGoHome := TRUE;
      "ST10Cylinder".Cy[35].Inout.AutoGoWork := FALSE;
      "ST10Cylinder".Cy[36].Inout.AutoGoHome := TRUE;
      "ST10Cylinder".Cy[36].Inout.AutoGoWork := FALSE;
      "ST10Cylinder".Cy[37].Inout.AutoGoHome := TRUE;
      "ST10Cylinder".Cy[37].Inout.AutoGoWork := FALSE;
      "ST10Cylinder".Cy[38].Inout.AutoGoHome := TRUE;
      "ST10Cylinder".Cy[38].Inout.AutoGoWork := FALSE;
      "ST10Cylinder".Cy[39].Inout.AutoGoHome := TRUE;
      "ST10Cylinder".Cy[39].Inout.AutoGoWork := FALSE;
    END_IF;
    IF tr_cond[116] THEN
      next_active[116] := FALSE;
      next_active[10] := TRUE;
    END_IF;
  END_IF;

  IF "DB_ST10_Flow26_JMagnetLoad_Unload_State".Flow.StepActive[117] THEN
    // Step 117: StoperReset_1
    IF NOT "DB_ST10_Flow26_JMagnetLoad_Unload_State".Flow.StepPrev[117] THEN
      "ST10Cylinder".Cy[33].Inout.AutoGoHome := TRUE;
      "ST10Cylinder".Cy[33].Inout.AutoGoWork := FALSE;
    END_IF;
    IF tr_cond[117] THEN
      next_active[117] := FALSE;
      next_active[237] := TRUE;
    END_IF;
  END_IF;

  IF "DB_ST10_Flow26_JMagnetLoad_Unload_State".Flow.StepActive[118] THEN
    // Step 118: StoperRelease_1
    IF NOT "DB_ST10_Flow26_JMagnetLoad_Unload_State".Flow.StepPrev[118] THEN
      "ST10Cylinder".Cy[33].Inout.AutoGoHome := FALSE;
      "ST10Cylinder".Cy[33].Inout.AutoGoWork := TRUE;
    END_IF;
    IF tr_cond[118] THEN
      next_active[118] := FALSE;
      next_active[37] := TRUE;
    END_IF;
  END_IF;

  IF "DB_ST10_Flow26_JMagnetLoad_Unload_State".Flow.StepActive[119] THEN
    // Step 119: AriveTimeDelay_1
    IF tr_cond[119] THEN
      next_active[119] := FALSE;
      next_active[117] := TRUE;
    END_IF;
  END_IF;

  IF "DB_ST10_Flow26_JMagnetLoad_Unload_State".Flow.StepActive[120] THEN
    // Step 120: AriveTimeDelay_2
    IF tr_cond[123] THEN
      next_active[120] := FALSE;
      next_active[121] := TRUE;
    END_IF;
  END_IF;

  IF "DB_ST10_Flow26_JMagnetLoad_Unload_State".Flow.StepActive[121] THEN
    // Step 121: StoperReset_2
    IF NOT "DB_ST10_Flow26_JMagnetLoad_Unload_State".Flow.StepPrev[121] THEN
      "ST10Cylinder".Cy[34].Inout.AutoGoHome := TRUE;
      "ST10Cylinder".Cy[34].Inout.AutoGoWork := FALSE;
    END_IF;
    IF tr_cond[124] THEN
      next_active[121] := FALSE;
      next_active[238] := TRUE;
    END_IF;
  END_IF;

  IF "DB_ST10_Flow26_JMagnetLoad_Unload_State".Flow.StepActive[122] THEN
    // Step 122: StoperRelease_2
    IF NOT "DB_ST10_Flow26_JMagnetLoad_Unload_State".Flow.StepPrev[122] THEN
      "ST10Cylinder".Cy[34].Inout.AutoGoHome := FALSE;
      "ST10Cylinder".Cy[34].Inout.AutoGoWork := TRUE;
    END_IF;
    IF tr_cond[125] THEN
      next_active[122] := FALSE;
      next_active[40] := TRUE;
    END_IF;
  END_IF;

  IF "DB_ST10_Flow26_JMagnetLoad_Unload_State".Flow.StepActive[123] THEN
    // Step 123: WaitPalletArive
    "DB_ST10_Flow26_JMagnetLoad_Unload_State".AutoProcessControl.Global.J.LoadStopRequestPallet_1 := TRUE;
    IF tr_cond[127] THEN
      next_active[123] := FALSE;
      next_active[124] := TRUE;
    END_IF;
  END_IF;

  IF "DB_ST10_Flow26_JMagnetLoad_Unload_State".Flow.StepActive[124] THEN
    // Step 124: TimeDelay
    IF tr_cond[128] THEN
      next_active[124] := FALSE;
      next_active[155] := TRUE;
    END_IF;
  END_IF;

  IF "DB_ST10_Flow26_JMagnetLoad_Unload_State".Flow.StepActive[125] THEN
    // Step 125: AriveTimeDelay_3
    IF tr_cond[129] THEN
      next_active[125] := FALSE;
      next_active[126] := TRUE;
    END_IF;
  END_IF;

  IF "DB_ST10_Flow26_JMagnetLoad_Unload_State".Flow.StepActive[126] THEN
    // Step 126: StoperReset_3
    IF NOT "DB_ST10_Flow26_JMagnetLoad_Unload_State".Flow.StepPrev[126] THEN
      "ST10Cylinder".Cy[35].Inout.AutoGoHome := TRUE;
      "ST10Cylinder".Cy[35].Inout.AutoGoWork := FALSE;
    END_IF;
    IF tr_cond[130] THEN
      next_active[126] := FALSE;
      next_active[239] := TRUE;
    END_IF;
  END_IF;

  IF "DB_ST10_Flow26_JMagnetLoad_Unload_State".Flow.StepActive[127] THEN
    // Step 127: StoperRelease_3
    IF NOT "DB_ST10_Flow26_JMagnetLoad_Unload_State".Flow.StepPrev[127] THEN
      "ST10Cylinder".Cy[35].Inout.AutoGoHome := FALSE;
      "ST10Cylinder".Cy[35].Inout.AutoGoWork := TRUE;
    END_IF;
    IF tr_cond[131] THEN
      next_active[127] := FALSE;
      next_active[44] := TRUE;
    END_IF;
  END_IF;

  IF "DB_ST10_Flow26_JMagnetLoad_Unload_State".Flow.StepActive[128] THEN
    // Step 128: WaitPalletArive_1
    "DB_ST10_Flow26_JMagnetLoad_Unload_State".AutoProcessControl.Global.J.LoadStopRequestPallet_2 := TRUE;
    IF tr_cond[133] THEN
      next_active[128] := FALSE;
      next_active[129] := TRUE;
    END_IF;
  END_IF;

  IF "DB_ST10_Flow26_JMagnetLoad_Unload_State".Flow.StepActive[129] THEN
    // Step 129: TimeDelay_1
    IF tr_cond[134] THEN
      next_active[129] := FALSE;
      next_active[156] := TRUE;
    END_IF;
  END_IF;

  IF "DB_ST10_Flow26_JMagnetLoad_Unload_State".Flow.StepActive[130] THEN
    // Step 130: AriveTimeDelay_4
    IF tr_cond[136] THEN
      next_active[130] := FALSE;
      next_active[131] := TRUE;
    END_IF;
  END_IF;

  IF "DB_ST10_Flow26_JMagnetLoad_Unload_State".Flow.StepActive[131] THEN
    // Step 131: StoperReset_4
    IF NOT "DB_ST10_Flow26_JMagnetLoad_Unload_State".Flow.StepPrev[131] THEN
      "ST10Cylinder".Cy[36].Inout.AutoGoHome := TRUE;
      "ST10Cylinder".Cy[36].Inout.AutoGoWork := FALSE;
    END_IF;
    IF tr_cond[137] THEN
      next_active[131] := FALSE;
      next_active[240] := TRUE;
    END_IF;
  END_IF;

  IF "DB_ST10_Flow26_JMagnetLoad_Unload_State".Flow.StepActive[132] THEN
    // Step 132: MotorStop
    IF NOT "DB_ST10_Flow26_JMagnetLoad_Unload_State".Flow.StepPrev[132] THEN
      "MotorControl".Dev[13].Auto.CCWStart := FALSE;
      "MotorControl".Dev[13].Auto.Start := FALSE;
      "MotorControl".Dev[14].Auto.CCWStart := FALSE;
      "MotorControl".Dev[14].Auto.Start := FALSE;
    END_IF;
    IF tr_cond[30] THEN
      next_active[132] := FALSE;
      next_active[116] := TRUE;
    END_IF;
  END_IF;

  IF "DB_ST10_Flow26_JMagnetLoad_Unload_State".Flow.StepActive[133] THEN
    // Step 133: StoperRelease_4
    IF NOT "DB_ST10_Flow26_JMagnetLoad_Unload_State".Flow.StepPrev[133] THEN
      "ST10Cylinder".Cy[36].Inout.AutoGoHome := FALSE;
      "ST10Cylinder".Cy[36].Inout.AutoGoWork := TRUE;
    END_IF;
    IF tr_cond[138] THEN
      next_active[133] := FALSE;
      next_active[48] := TRUE;
    END_IF;
  END_IF;

  IF "DB_ST10_Flow26_JMagnetLoad_Unload_State".Flow.StepActive[134] THEN
    // Step 134: WaitPalletArive_2
    "DB_ST10_Flow26_JMagnetLoad_Unload_State".AutoProcessControl.Global.J.LoadStopRequestPallet_3 := TRUE;
    IF tr_cond[140] THEN
      next_active[134] := FALSE;
      next_active[135] := TRUE;
    END_IF;
  END_IF;

  IF "DB_ST10_Flow26_JMagnetLoad_Unload_State".Flow.StepActive[135] THEN
    // Step 135: TimeDelay_2
    IF tr_cond[144] THEN
      next_active[135] := FALSE;
      next_active[157] := TRUE;
    END_IF;
  END_IF;

  IF "DB_ST10_Flow26_JMagnetLoad_Unload_State".Flow.StepActive[136] THEN
    // Step 136: AriveTimeDelay_5
    IF tr_cond[145] THEN
      next_active[136] := FALSE;
      next_active[137] := TRUE;
    END_IF;
  END_IF;

  IF "DB_ST10_Flow26_JMagnetLoad_Unload_State".Flow.StepActive[137] THEN
    // Step 137: StoperReset_5
    IF NOT "DB_ST10_Flow26_JMagnetLoad_Unload_State".Flow.StepPrev[137] THEN
      "ST10Cylinder".Cy[37].Inout.AutoGoHome := TRUE;
      "ST10Cylinder".Cy[37].Inout.AutoGoWork := FALSE;
    END_IF;
    IF tr_cond[146] THEN
      next_active[137] := FALSE;
      next_active[241] := TRUE;
    END_IF;
  END_IF;

  IF "DB_ST10_Flow26_JMagnetLoad_Unload_State".Flow.StepActive[138] THEN
    // Step 138: StoperRelease_5
    IF NOT "DB_ST10_Flow26_JMagnetLoad_Unload_State".Flow.StepPrev[138] THEN
      "ST10Cylinder".Cy[37].Inout.AutoGoHome := FALSE;
      "ST10Cylinder".Cy[37].Inout.AutoGoWork := TRUE;
    END_IF;
    IF tr_cond[147] THEN
      next_active[138] := FALSE;
      next_active[52] := TRUE;
    END_IF;
  END_IF;

  IF "DB_ST10_Flow26_JMagnetLoad_Unload_State".Flow.StepActive[139] THEN
    // Step 139: WaitPalletArive_3
    "DB_ST10_Flow26_JMagnetLoad_Unload_State".AutoProcessControl.Global.J.EmptyStopRequestPallet_1 := TRUE;
    IF tr_cond[149] THEN
      next_active[139] := FALSE;
      next_active[140] := TRUE;
    END_IF;
  END_IF;

  IF "DB_ST10_Flow26_JMagnetLoad_Unload_State".Flow.StepActive[140] THEN
    // Step 140: TimeDelay_3
    IF tr_cond[150] THEN
      next_active[140] := FALSE;
      next_active[201] := TRUE;
    END_IF;
  END_IF;

  IF "DB_ST10_Flow26_JMagnetLoad_Unload_State".Flow.StepActive[141] THEN
    // Step 141: AriveTimeDelay_6
    IF tr_cond[151] THEN
      next_active[141] := FALSE;
      next_active[144] := TRUE;
    END_IF;
  END_IF;

  IF "DB_ST10_Flow26_JMagnetLoad_Unload_State".Flow.StepActive[142] THEN
    // Step 142: LoadingStop_1
    IF tr_cond[141] THEN
      next_active[142] := FALSE;
      next_active[31] := TRUE;
    END_IF;
  END_IF;

  IF "DB_ST10_Flow26_JMagnetLoad_Unload_State".Flow.StepActive[143] THEN
    // Step 143: Step143
  END_IF;

  IF "DB_ST10_Flow26_JMagnetLoad_Unload_State".Flow.StepActive[144] THEN
    // Step 144: StoperReset_6
    IF NOT "DB_ST10_Flow26_JMagnetLoad_Unload_State".Flow.StepPrev[144] THEN
      "ST10Cylinder".Cy[38].Inout.AutoGoHome := TRUE;
      "ST10Cylinder".Cy[38].Inout.AutoGoWork := FALSE;
    END_IF;
    IF tr_cond[152] THEN
      next_active[144] := FALSE;
      next_active[242] := TRUE;
    END_IF;
  END_IF;

  IF "DB_ST10_Flow26_JMagnetLoad_Unload_State".Flow.StepActive[145] THEN
    // Step 145: StoperRelease_6
    IF NOT "DB_ST10_Flow26_JMagnetLoad_Unload_State".Flow.StepPrev[145] THEN
      "ST10Cylinder".Cy[38].Inout.AutoGoHome := FALSE;
      "ST10Cylinder".Cy[38].Inout.AutoGoWork := TRUE;
    END_IF;
    IF tr_cond[153] THEN
      next_active[145] := FALSE;
      next_active[56] := TRUE;
    END_IF;
  END_IF;

  IF "DB_ST10_Flow26_JMagnetLoad_Unload_State".Flow.StepActive[146] THEN
    // Step 146: WaitPalletArive_4
    "DB_ST10_Flow26_JMagnetLoad_Unload_State".AutoProcessControl.Global.J.EmptyStopRequestPallet_2 := TRUE;
    IF tr_cond[155] THEN
      next_active[146] := FALSE;
      next_active[147] := TRUE;
    END_IF;
  END_IF;

  IF "DB_ST10_Flow26_JMagnetLoad_Unload_State".Flow.StepActive[147] THEN
    // Step 147: TimeDelay_4
    IF tr_cond[156] THEN
      next_active[147] := FALSE;
      next_active[202] := TRUE;
    END_IF;
  END_IF;

  IF "DB_ST10_Flow26_JMagnetLoad_Unload_State".Flow.StepActive[148] THEN
    // Step 148: AriveTimeDelay_7
    IF tr_cond[157] THEN
      next_active[148] := FALSE;
      next_active[149] := TRUE;
    END_IF;
  END_IF;

  IF "DB_ST10_Flow26_JMagnetLoad_Unload_State".Flow.StepActive[149] THEN
    // Step 149: StoperReset_7
    IF NOT "DB_ST10_Flow26_JMagnetLoad_Unload_State".Flow.StepPrev[149] THEN
      "ST10Cylinder".Cy[39].Inout.AutoGoHome := TRUE;
      "ST10Cylinder".Cy[39].Inout.AutoGoWork := FALSE;
    END_IF;
    IF tr_cond[158] THEN
      next_active[149] := FALSE;
      next_active[243] := TRUE;
    END_IF;
  END_IF;

  IF "DB_ST10_Flow26_JMagnetLoad_Unload_State".Flow.StepActive[150] THEN
    // Step 150: StoperRelease_7
    IF NOT "DB_ST10_Flow26_JMagnetLoad_Unload_State".Flow.StepPrev[150] THEN
      "ST10Cylinder".Cy[39].Inout.AutoGoHome := FALSE;
      "ST10Cylinder".Cy[39].Inout.AutoGoWork := TRUE;
    END_IF;
    IF tr_cond[159] THEN
      next_active[150] := FALSE;
      next_active[60] := TRUE;
    END_IF;
  END_IF;

  IF "DB_ST10_Flow26_JMagnetLoad_Unload_State".Flow.StepActive[151] THEN
    // Step 151: WaitPalletArive_5
    "DB_ST10_Flow26_JMagnetLoad_Unload_State".AutoProcessControl.Global.J.EmptyStopRequestPallet_3 := TRUE;
    IF tr_cond[161] THEN
      next_active[151] := FALSE;
      next_active[152] := TRUE;
    END_IF;
  END_IF;

  IF "DB_ST10_Flow26_JMagnetLoad_Unload_State".Flow.StepActive[152] THEN
    // Step 152: TimeDelay_5
    IF tr_cond[162] THEN
      next_active[152] := FALSE;
      next_active[203] := TRUE;
    END_IF;
  END_IF;

  IF "DB_ST10_Flow26_JMagnetLoad_Unload_State".Flow.StepActive[153] THEN
    // Step 153: Step153
    IF tr_cond[163] THEN
      next_active[153] := FALSE;
      next_active[178] := TRUE;
    END_IF;
  END_IF;

  IF "DB_ST10_Flow26_JMagnetLoad_Unload_State".Flow.StepActive[154] THEN
    // Step 154: CheckMachine Mode_1
    IF tr_cond[164] THEN
      next_active[154] := FALSE;
      next_active[142] := TRUE;
    END_IF;
  END_IF;

  IF "DB_ST10_Flow26_JMagnetLoad_Unload_State".Flow.StepActive[155] THEN
    // Step 155: CheckMachine Mode_2
    IF tr_cond[165] THEN
      next_active[155] := FALSE;
      next_active[28] := TRUE;
    END_IF;
  END_IF;

  IF "DB_ST10_Flow26_JMagnetLoad_Unload_State".Flow.StepActive[156] THEN
    // Step 156: CheckMachine Mode_3
    IF tr_cond[166] THEN
      next_active[156] := FALSE;
      next_active[29] := TRUE;
    END_IF;
  END_IF;

  IF "DB_ST10_Flow26_JMagnetLoad_Unload_State".Flow.StepActive[157] THEN
    // Step 157: CheckMachine Mode_4
    IF tr_cond[167] THEN
      next_active[157] := FALSE;
      next_active[30] := TRUE;
    END_IF;
  END_IF;

  IF "DB_ST10_Flow26_JMagnetLoad_Unload_State".Flow.StepActive[158] THEN
    // Step 158: CheckMachine Mode_5
    IF tr_cond[196] THEN
      next_active[158] := FALSE;
      next_active[63] := TRUE;
    END_IF;
  END_IF;

  IF "DB_ST10_Flow26_JMagnetLoad_Unload_State".Flow.StepActive[159] THEN
    // Step 159: AriveTimeDelay_8
    IF tr_cond[168] THEN
      next_active[159] := FALSE;
      next_active[161] := TRUE;
    END_IF;
  END_IF;

  IF "DB_ST10_Flow26_JMagnetLoad_Unload_State".Flow.StepActive[160] THEN
    // Step 160: LoadStop_11
    IF tr_cond[172] THEN
      next_active[160] := FALSE;
      next_active[64] := TRUE;
    END_IF;
  END_IF;

  IF "DB_ST10_Flow26_JMagnetLoad_Unload_State".Flow.StepActive[161] THEN
    // Step 161: StoperReset_8
    IF NOT "DB_ST10_Flow26_JMagnetLoad_Unload_State".Flow.StepPrev[161] THEN
      "ST10Cylinder".Cy[33].Inout.AutoGoHome := TRUE;
      "ST10Cylinder".Cy[33].Inout.AutoGoWork := FALSE;
    END_IF;
    IF tr_cond[173] THEN
      next_active[161] := FALSE;
      next_active[244] := TRUE;
    END_IF;
  END_IF;

  IF "DB_ST10_Flow26_JMagnetLoad_Unload_State".Flow.StepActive[162] THEN
    // Step 162: StoperRelease_8
    IF NOT "DB_ST10_Flow26_JMagnetLoad_Unload_State".Flow.StepPrev[162] THEN
      "ST10Cylinder".Cy[33].Inout.AutoGoHome := FALSE;
      "ST10Cylinder".Cy[33].Inout.AutoGoWork := TRUE;
    END_IF;
    IF tr_cond[174] THEN
      next_active[162] := FALSE;
      next_active[67] := TRUE;
    END_IF;
  END_IF;

  IF "DB_ST10_Flow26_JMagnetLoad_Unload_State".Flow.StepActive[163] THEN
    // Step 163: AriveTimeDelay_9
    IF tr_cond[176] THEN
      next_active[163] := FALSE;
      next_active[164] := TRUE;
    END_IF;
  END_IF;

  IF "DB_ST10_Flow26_JMagnetLoad_Unload_State".Flow.StepActive[164] THEN
    // Step 164: StoperReset_9
    IF NOT "DB_ST10_Flow26_JMagnetLoad_Unload_State".Flow.StepPrev[164] THEN
      "ST10Cylinder".Cy[34].Inout.AutoGoHome := TRUE;
      "ST10Cylinder".Cy[34].Inout.AutoGoWork := FALSE;
    END_IF;
    IF tr_cond[177] THEN
      next_active[164] := FALSE;
      next_active[245] := TRUE;
    END_IF;
  END_IF;

  IF "DB_ST10_Flow26_JMagnetLoad_Unload_State".Flow.StepActive[165] THEN
    // Step 165: StoperRelease_9
    IF NOT "DB_ST10_Flow26_JMagnetLoad_Unload_State".Flow.StepPrev[165] THEN
      "ST10Cylinder".Cy[34].Inout.AutoGoHome := FALSE;
      "ST10Cylinder".Cy[34].Inout.AutoGoWork := TRUE;
    END_IF;
    IF tr_cond[178] THEN
      next_active[165] := FALSE;
      next_active[71] := TRUE;
    END_IF;
  END_IF;

  IF "DB_ST10_Flow26_JMagnetLoad_Unload_State".Flow.StepActive[166] THEN
    // Step 166: WaitPalletArive_6
    "DB_ST10_Flow26_JMagnetLoad_Unload_State".AutoProcessControl.Global.J.LoadStopRequestPallet_3 := TRUE;
    IF tr_cond[180] THEN
      next_active[166] := FALSE;
      next_active[167] := TRUE;
    END_IF;
  END_IF;

  IF "DB_ST10_Flow26_JMagnetLoad_Unload_State".Flow.StepActive[167] THEN
    // Step 167: TimeDelay_6
    IF tr_cond[181] THEN
      next_active[167] := FALSE;
      next_active[179] := TRUE;
    END_IF;
  END_IF;

  IF "DB_ST10_Flow26_JMagnetLoad_Unload_State".Flow.StepActive[168] THEN
    // Step 168: AriveTimeDelay_10
    IF tr_cond[182] THEN
      next_active[168] := FALSE;
      next_active[169] := TRUE;
    END_IF;
  END_IF;

  IF "DB_ST10_Flow26_JMagnetLoad_Unload_State".Flow.StepActive[169] THEN
    // Step 169: StoperReset_10
    IF NOT "DB_ST10_Flow26_JMagnetLoad_Unload_State".Flow.StepPrev[169] THEN
      "ST10Cylinder".Cy[35].Inout.AutoGoHome := TRUE;
      "ST10Cylinder".Cy[35].Inout.AutoGoWork := FALSE;
    END_IF;
    IF tr_cond[183] THEN
      next_active[169] := FALSE;
      next_active[246] := TRUE;
    END_IF;
  END_IF;

  IF "DB_ST10_Flow26_JMagnetLoad_Unload_State".Flow.StepActive[170] THEN
    // Step 170: StoperRelease_10
    IF NOT "DB_ST10_Flow26_JMagnetLoad_Unload_State".Flow.StepPrev[170] THEN
      "ST10Cylinder".Cy[35].Inout.AutoGoHome := FALSE;
      "ST10Cylinder".Cy[35].Inout.AutoGoWork := TRUE;
    END_IF;
    IF tr_cond[184] THEN
      next_active[170] := FALSE;
      next_active[75] := TRUE;
    END_IF;
  END_IF;

  IF "DB_ST10_Flow26_JMagnetLoad_Unload_State".Flow.StepActive[171] THEN
    // Step 171: WaitPalletArive_7
    "DB_ST10_Flow26_JMagnetLoad_Unload_State".AutoProcessControl.Global.J.LoadStopRequestPallet_4 := TRUE;
    IF tr_cond[186] THEN
      next_active[171] := FALSE;
      next_active[172] := TRUE;
    END_IF;
  END_IF;

  IF "DB_ST10_Flow26_JMagnetLoad_Unload_State".Flow.StepActive[172] THEN
    // Step 172: TimeDelay_7
    IF tr_cond[187] THEN
      next_active[172] := FALSE;
      next_active[158] := TRUE;
    END_IF;
  END_IF;

  IF "DB_ST10_Flow26_JMagnetLoad_Unload_State".Flow.StepActive[173] THEN
    // Step 173: AriveTimeDelay_11
    IF tr_cond[188] THEN
      next_active[173] := FALSE;
      next_active[174] := TRUE;
    END_IF;
  END_IF;

  IF "DB_ST10_Flow26_JMagnetLoad_Unload_State".Flow.StepActive[174] THEN
    // Step 174: StoperReset_11
    IF NOT "DB_ST10_Flow26_JMagnetLoad_Unload_State".Flow.StepPrev[174] THEN
      "ST10Cylinder".Cy[36].Inout.AutoGoHome := TRUE;
      "ST10Cylinder".Cy[36].Inout.AutoGoWork := FALSE;
    END_IF;
    IF tr_cond[189] THEN
      next_active[174] := FALSE;
      next_active[247] := TRUE;
    END_IF;
  END_IF;

  IF "DB_ST10_Flow26_JMagnetLoad_Unload_State".Flow.StepActive[175] THEN
    // Step 175: StoperRelease_11
    IF NOT "DB_ST10_Flow26_JMagnetLoad_Unload_State".Flow.StepPrev[175] THEN
      "ST10Cylinder".Cy[36].Inout.AutoGoHome := FALSE;
      "ST10Cylinder".Cy[36].Inout.AutoGoWork := TRUE;
    END_IF;
    IF tr_cond[190] THEN
      next_active[175] := FALSE;
      next_active[79] := TRUE;
    END_IF;
  END_IF;

  IF "DB_ST10_Flow26_JMagnetLoad_Unload_State".Flow.StepActive[176] THEN
    // Step 176: WaitPalletArive_8
    IF tr_cond[192] THEN
      next_active[176] := FALSE;
      next_active[177] := TRUE;
    END_IF;
  END_IF;

  IF "DB_ST10_Flow26_JMagnetLoad_Unload_State".Flow.StepActive[177] THEN
    // Step 177: TimeDelay_8
    IF tr_cond[193] THEN
      next_active[177] := FALSE;
      next_active[180] := TRUE;
    END_IF;
  END_IF;

  IF "DB_ST10_Flow26_JMagnetLoad_Unload_State".Flow.StepActive[178] THEN
    // Step 178: CheckMachine Mode_6
    IF tr_cond[194] THEN
      next_active[178] := FALSE;
      next_active[160] := TRUE;
    END_IF;
  END_IF;

  IF "DB_ST10_Flow26_JMagnetLoad_Unload_State".Flow.StepActive[179] THEN
    // Step 179: CheckMachine Mode_7
    IF tr_cond[195] THEN
      next_active[179] := FALSE;
      next_active[62] := TRUE;
    END_IF;
  END_IF;

  IF "DB_ST10_Flow26_JMagnetLoad_Unload_State".Flow.StepActive[180] THEN
    // Step 180: CheckMachine Mode_8
    IF tr_cond[171] THEN
      next_active[180] := FALSE;
      next_active[61] := TRUE;
    END_IF;
  END_IF;

  IF "DB_ST10_Flow26_JMagnetLoad_Unload_State".Flow.StepActive[181] THEN
    // Step 181: WaitAllStoperReset
    IF tr_cond[197] THEN
      next_active[181] := FALSE;
      next_active[80] := TRUE;
    END_IF;
  END_IF;

  IF "DB_ST10_Flow26_JMagnetLoad_Unload_State".Flow.StepActive[182] THEN
    // Step 182: Step182
    IF tr_cond[198] THEN
      next_active[182] := FALSE;
    END_IF;
  END_IF;

  IF "DB_ST10_Flow26_JMagnetLoad_Unload_State".Flow.StepActive[183] THEN
    // Step 183: WaitPalletArive_9
    "DB_ST10_Flow26_JMagnetLoad_Unload_State".AutoProcessControl.Global.J.LoadStopRequestPallet_2 := TRUE;
    IF tr_cond[199] THEN
      next_active[183] := FALSE;
      next_active[184] := TRUE;
    END_IF;
  END_IF;

  IF "DB_ST10_Flow26_JMagnetLoad_Unload_State".Flow.StepActive[184] THEN
    // Step 184: TimeDelay_9
    IF tr_cond[201] THEN
      next_active[184] := FALSE;
      next_active[178] := TRUE;
    END_IF;
  END_IF;

  IF "DB_ST10_Flow26_JMagnetLoad_Unload_State".Flow.StepActive[200] THEN
    // Step 200: CheckMachineMode
    IF tr_cond[200] THEN
      next_active[200] := FALSE;
      next_active[181] := TRUE;
    END_IF;
  END_IF;

  IF "DB_ST10_Flow26_JMagnetLoad_Unload_State".Flow.StepActive[201] THEN
    // Step 201: UnloadStoper_1
    IF tr_cond[135] THEN
      next_active[201] := FALSE;
      next_active[49] := TRUE;
    END_IF;
  END_IF;

  IF "DB_ST10_Flow26_JMagnetLoad_Unload_State".Flow.StepActive[202] THEN
    // Step 202: UnloadStoper_2
    IF tr_cond[202] THEN
      next_active[202] := FALSE;
      next_active[53] := TRUE;
    END_IF;
  END_IF;

  IF "DB_ST10_Flow26_JMagnetLoad_Unload_State".Flow.StepActive[203] THEN
    // Step 203: UnloadStoper_3
    IF tr_cond[203] THEN
      next_active[203] := FALSE;
      next_active[57] := TRUE;
    END_IF;
  END_IF;

  IF "DB_ST10_Flow26_JMagnetLoad_Unload_State".Flow.StepActive[237] THEN
    // Step 237: Process Finish_1
    IF tr_cond[249] THEN
      next_active[237] := FALSE;
      next_active[154] := TRUE;
    END_IF;
  END_IF;

  IF "DB_ST10_Flow26_JMagnetLoad_Unload_State".Flow.StepActive[238] THEN
    // Step 238: Process Finish_2
    IF tr_cond[250] THEN
      next_active[238] := FALSE;
      next_active[155] := TRUE;
    END_IF;
  END_IF;

  IF "DB_ST10_Flow26_JMagnetLoad_Unload_State".Flow.StepActive[239] THEN
    // Step 239: Process Finish_3
    IF tr_cond[251] THEN
      next_active[239] := FALSE;
      next_active[156] := TRUE;
    END_IF;
  END_IF;

  IF "DB_ST10_Flow26_JMagnetLoad_Unload_State".Flow.StepActive[240] THEN
    // Step 240: Process Finish_4
    IF tr_cond[252] THEN
      next_active[240] := FALSE;
      next_active[157] := TRUE;
    END_IF;
  END_IF;

  IF "DB_ST10_Flow26_JMagnetLoad_Unload_State".Flow.StepActive[241] THEN
    // Step 241: Process Finish_5
    IF tr_cond[253] THEN
      next_active[241] := FALSE;
      next_active[201] := TRUE;
    END_IF;
  END_IF;

  IF "DB_ST10_Flow26_JMagnetLoad_Unload_State".Flow.StepActive[242] THEN
    // Step 242: Process Finish_6
    IF tr_cond[254] THEN
      next_active[242] := FALSE;
      next_active[202] := TRUE;
    END_IF;
  END_IF;

  IF "DB_ST10_Flow26_JMagnetLoad_Unload_State".Flow.StepActive[243] THEN
    // Step 243: Process Finish_7
    IF tr_cond[255] THEN
      next_active[243] := FALSE;
      next_active[203] := TRUE;
    END_IF;
  END_IF;

  IF "DB_ST10_Flow26_JMagnetLoad_Unload_State".Flow.StepActive[244] THEN
    // Step 244: Process Finish_8
    IF tr_cond[256] THEN
      next_active[244] := FALSE;
      next_active[153] := TRUE;
    END_IF;
  END_IF;

  IF "DB_ST10_Flow26_JMagnetLoad_Unload_State".Flow.StepActive[245] THEN
    // Step 245: Process Finish_9
    IF tr_cond[257] THEN
      next_active[245] := FALSE;
      next_active[179] := TRUE;
    END_IF;
  END_IF;

  IF "DB_ST10_Flow26_JMagnetLoad_Unload_State".Flow.StepActive[246] THEN
    // Step 246: Process Finish_10
    IF tr_cond[258] THEN
      next_active[246] := FALSE;
      next_active[158] := TRUE;
    END_IF;
  END_IF;

  IF "DB_ST10_Flow26_JMagnetLoad_Unload_State".Flow.StepActive[247] THEN
    // Step 247: Process Finish_11
    IF tr_cond[259] THEN
      next_active[247] := FALSE;
      next_active[180] := TRUE;
    END_IF;
  END_IF;

  FOR idx := 1 TO 247 DO
    "DB_ST10_Flow26_JMagnetLoad_Unload_State".Flow.StepPrev[idx] := "DB_ST10_Flow26_JMagnetLoad_Unload_State".Flow.StepActive[idx];
    "DB_ST10_Flow26_JMagnetLoad_Unload_State".Flow.StepActive[idx] := next_active[idx];
  END_FOR;
END_FUNCTION